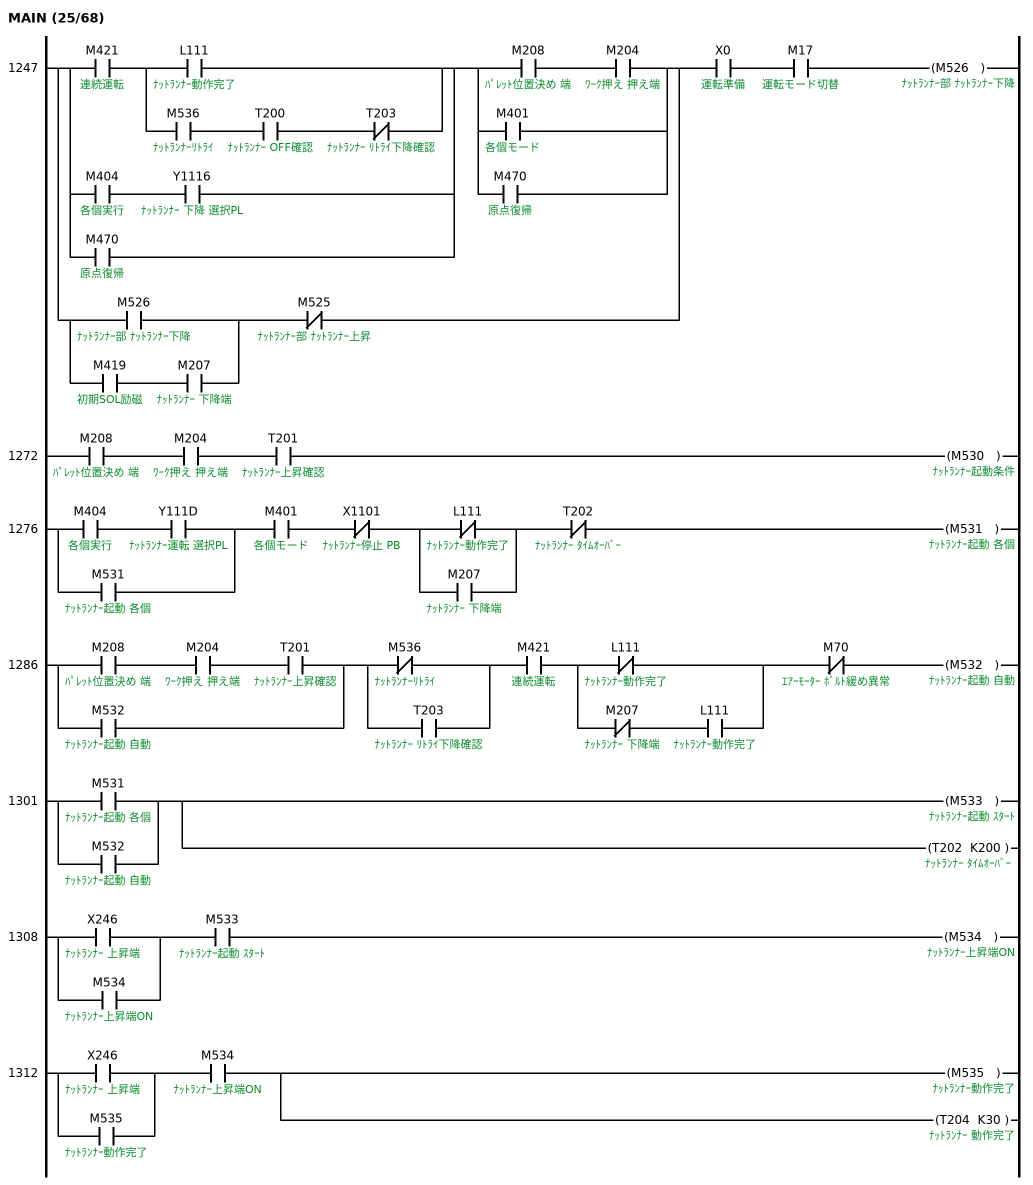
[picture p24: ladder of MAIN, rungs at steps 1247 to 1312]
1247  LD      M421  ; 連続運転
      LD      L111  ; ﾅｯﾄﾗﾝﾅｰ動作完了
      LD      M536  ; ﾅｯﾄﾗﾝﾅｰﾘﾄﾗｲ
      AND     T200  ; ﾅｯﾄﾗﾝﾅｰ OFF確認
      ANI     T203  ; ﾅｯﾄﾗﾝﾅｰ ﾘﾄﾗｲ下降確認
      ORB
      ANB
      LD      M404  ; 各個実行
      AND     Y1116  ; ﾅｯﾄﾗﾝﾅｰ 下降 選択PL
      ORB
      OR      M470  ; 原点復帰
      LD      M208  ; ﾊﾟﾚｯﾄ位置決め 端
      AND     M204  ; ﾜｰｸ押え 押え端
      OR      M401  ; 各個モード
      OR      M470  ; 原点復帰
      ANB
      LD      M526  ; ﾅｯﾄﾗﾝﾅｰ部 ﾅｯﾄﾗﾝﾅｰ下降
      LD      M419  ; 初期SOL励磁
      AND     M207  ; ﾅｯﾄﾗﾝﾅｰ 下降端
      ORB
      ANI     M525  ; ﾅｯﾄﾗﾝﾅｰ部 ﾅｯﾄﾗﾝﾅｰ上昇
      ORB
      AND     X0  ; 運転準備
      AND     M17  ; 運転モード切替
      OUT     M526  ; ﾅｯﾄﾗﾝﾅｰ部 ﾅｯﾄﾗﾝﾅｰ下降
1272  LD      M208  ; ﾊﾟﾚｯﾄ位置決め 端
      AND     M204  ; ﾜｰｸ押え 押え端
      AND     T201  ; ﾅｯﾄﾗﾝﾅｰ上昇確認
      OUT     M530  ; ﾅｯﾄﾗﾝﾅｰ起動条件
1276  LD      M404  ; 各個実行
      AND     Y111D  ; ﾅｯﾄﾗﾝﾅｰ運転 選択PL
      OR      M531  ; ﾅｯﾄﾗﾝﾅｰ起動 各個
      AND     M401  ; 各個モード
      ANI     X1101  ; ﾅｯﾄﾗﾝﾅｰ停止 PB
      LDI     L111  ; ﾅｯﾄﾗﾝﾅｰ動作完了
      OR      M207  ; ﾅｯﾄﾗﾝﾅｰ 下降端
      ANB
      ANI     T202  ; ﾅｯﾄﾗﾝﾅｰ ﾀｲﾑｵｰﾊﾞｰ
      OUT     M531  ; ﾅｯﾄﾗﾝﾅｰ起動 各個
1286  LD      M208  ; ﾊﾟﾚｯﾄ位置決め 端
      AND     M204  ; ﾜｰｸ押え 押え端
      AND     T201  ; ﾅｯﾄﾗﾝﾅｰ上昇確認
      OR      M532  ; ﾅｯﾄﾗﾝﾅｰ起動 自動
      LDI     M536  ; ﾅｯﾄﾗﾝﾅｰﾘﾄﾗｲ
      OR      T203  ; ﾅｯﾄﾗﾝﾅｰ ﾘﾄﾗｲ下降確認
      ANB
      AND     M421  ; 連続運転
      LDI     L111  ; ﾅｯﾄﾗﾝﾅｰ動作完了
      LDI     M207  ; ﾅｯﾄﾗﾝﾅｰ 下降端
      AND     L111  ; ﾅｯﾄﾗﾝﾅｰ動作完了
      ORB
      ANB
      ANI     M70  ; ｴｱｰﾓｰﾀｰ ﾎﾞﾙﾄ緩め異常
      OUT     M532  ; ﾅｯﾄﾗﾝﾅｰ起動 自動
1301  LD      M531  ; ﾅｯﾄﾗﾝﾅｰ起動 各個
      OR      M532  ; ﾅｯﾄﾗﾝﾅｰ起動 自動
      OUT     M533  ; ﾅｯﾄﾗﾝﾅｰ起動 ｽﾀｰﾄ
      OUT     T202 K200  ; ﾅｯﾄﾗﾝﾅｰ ﾀｲﾑｵｰﾊﾞｰ
1308  LD      X246  ; ﾅｯﾄﾗﾝﾅｰ 上昇端
      OR      M534  ; ﾅｯﾄﾗﾝﾅｰ上昇端ON
      AND     M533  ; ﾅｯﾄﾗﾝﾅｰ起動 ｽﾀｰﾄ
      OUT     M534  ; ﾅｯﾄﾗﾝﾅｰ上昇端ON
1312  LD      X246  ; ﾅｯﾄﾗﾝﾅｰ 上昇端
      OR      M535  ; ﾅｯﾄﾗﾝﾅｰ動作完了
      AND     M534  ; ﾅｯﾄﾗﾝﾅｰ上昇端ON
      OUT     M535  ; ﾅｯﾄﾗﾝﾅｰ動作完了
      OUT     T204 K30  ; ﾅｯﾄﾗﾝﾅｰ 動作完了
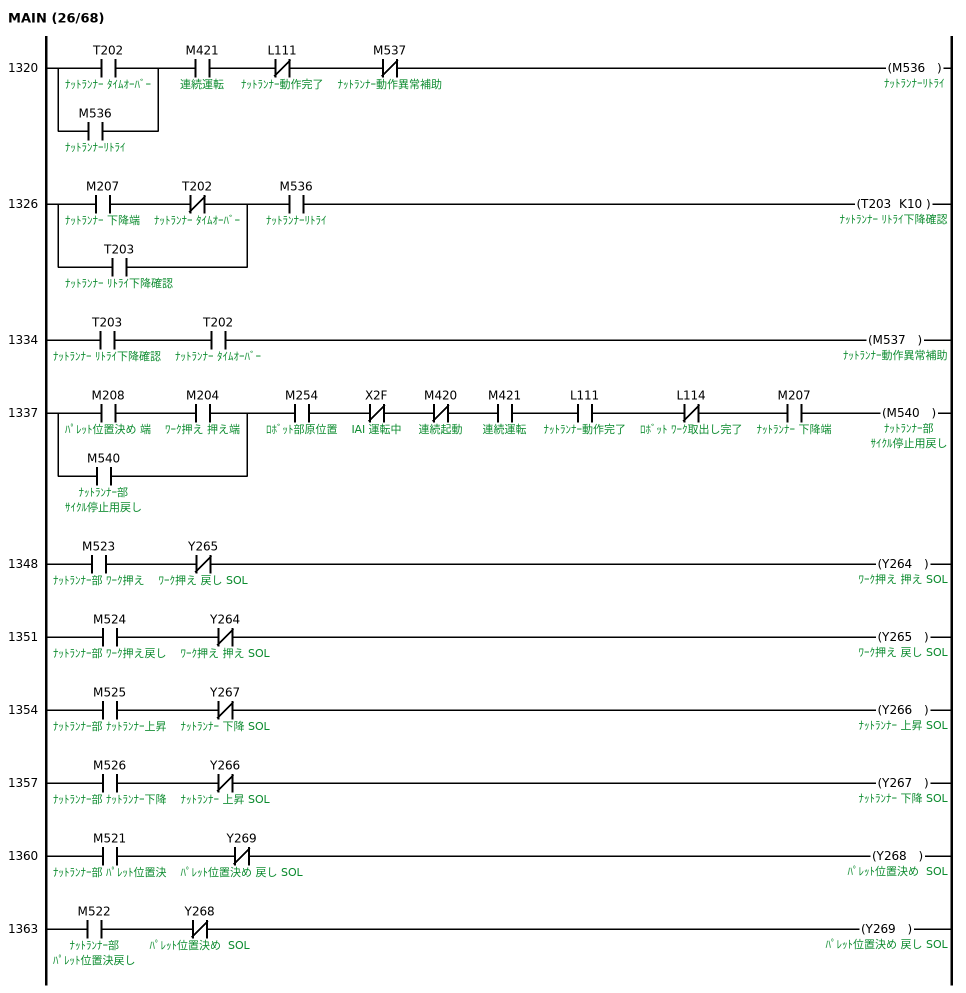
1320  LD      T202  ; ﾅｯﾄﾗﾝﾅｰ ﾀｲﾑｵｰﾊﾞｰ
      OR      M536  ; ﾅｯﾄﾗﾝﾅｰﾘﾄﾗｲ
      AND     M421  ; 連続運転
      ANI     L111  ; ﾅｯﾄﾗﾝﾅｰ動作完了
      ANI     M537  ; ﾅｯﾄﾗﾝﾅｰ動作異常補助
      OUT     M536  ; ﾅｯﾄﾗﾝﾅｰﾘﾄﾗｲ
1326  LD      M207  ; ﾅｯﾄﾗﾝﾅｰ 下降端
      ANI     T202  ; ﾅｯﾄﾗﾝﾅｰ ﾀｲﾑｵｰﾊﾞｰ
      OR      T203  ; ﾅｯﾄﾗﾝﾅｰ ﾘﾄﾗｲ下降確認
      AND     M536  ; ﾅｯﾄﾗﾝﾅｰﾘﾄﾗｲ
      OUT     T203 K10  ; ﾅｯﾄﾗﾝﾅｰ ﾘﾄﾗｲ下降確認
1334  LD      T203  ; ﾅｯﾄﾗﾝﾅｰ ﾘﾄﾗｲ下降確認
      AND     T202  ; ﾅｯﾄﾗﾝﾅｰ ﾀｲﾑｵｰﾊﾞｰ
      OUT     M537  ; ﾅｯﾄﾗﾝﾅｰ動作異常補助
1337  LD      M208  ; ﾊﾟﾚｯﾄ位置決め 端
      AND     M204  ; ﾜｰｸ押え 押え端
      OR      M540  ; ﾅｯﾄﾗﾝﾅｰ部 ｻｲｸﾙ停止用戻し
      AND     M254  ; ﾛﾎﾞｯﾄ部原位置
      ANI     X2F  ; IAI 運転中
      ANI     M420  ; 連続起動
      AND     M421  ; 連続運転
      AND     L111  ; ﾅｯﾄﾗﾝﾅｰ動作完了
      ANI     L114  ; ﾛﾎﾞｯﾄ ﾜｰｸ取出し完了
      AND     M207  ; ﾅｯﾄﾗﾝﾅｰ 下降端
      OUT     M540  ; ﾅｯﾄﾗﾝﾅｰ部 ｻｲｸﾙ停止用戻し
1348  LD      M523  ; ﾅｯﾄﾗﾝﾅｰ部 ﾜｰｸ押え
      ANI     Y265  ; ﾜｰｸ押え 戻し SOL
      OUT     Y264  ; ﾜｰｸ押え 押え SOL
1351  LD      M524  ; ﾅｯﾄﾗﾝﾅｰ部 ﾜｰｸ押え戻し
      ANI     Y264  ; ﾜｰｸ押え 押え SOL
      OUT     Y265  ; ﾜｰｸ押え 戻し SOL
1354  LD      M525  ; ﾅｯﾄﾗﾝﾅｰ部 ﾅｯﾄﾗﾝﾅｰ上昇
      ANI     Y267  ; ﾅｯﾄﾗﾝﾅｰ 下降 SOL
      OUT     Y266  ; ﾅｯﾄﾗﾝﾅｰ 上昇 SOL
1357  LD      M526  ; ﾅｯﾄﾗﾝﾅｰ部 ﾅｯﾄﾗﾝﾅｰ下降
      ANI     Y266  ; ﾅｯﾄﾗﾝﾅｰ 上昇 SOL
      OUT     Y267  ; ﾅｯﾄﾗﾝﾅｰ 下降 SOL
1360  LD      M521  ; ﾅｯﾄﾗﾝﾅｰ部 ﾊﾟﾚｯﾄ位置決
      ANI     Y269  ; ﾊﾟﾚｯﾄ位置決め 戻し SOL
      OUT     Y268  ; ﾊﾟﾚｯﾄ位置決め  SOL
1363  LD      M522  ; ﾅｯﾄﾗﾝﾅｰ部 ﾊﾟﾚｯﾄ位置決戻し
      ANI     Y268  ; ﾊﾟﾚｯﾄ位置決め  SOL
      OUT     Y269  ; ﾊﾟﾚｯﾄ位置決め 戻し SOL
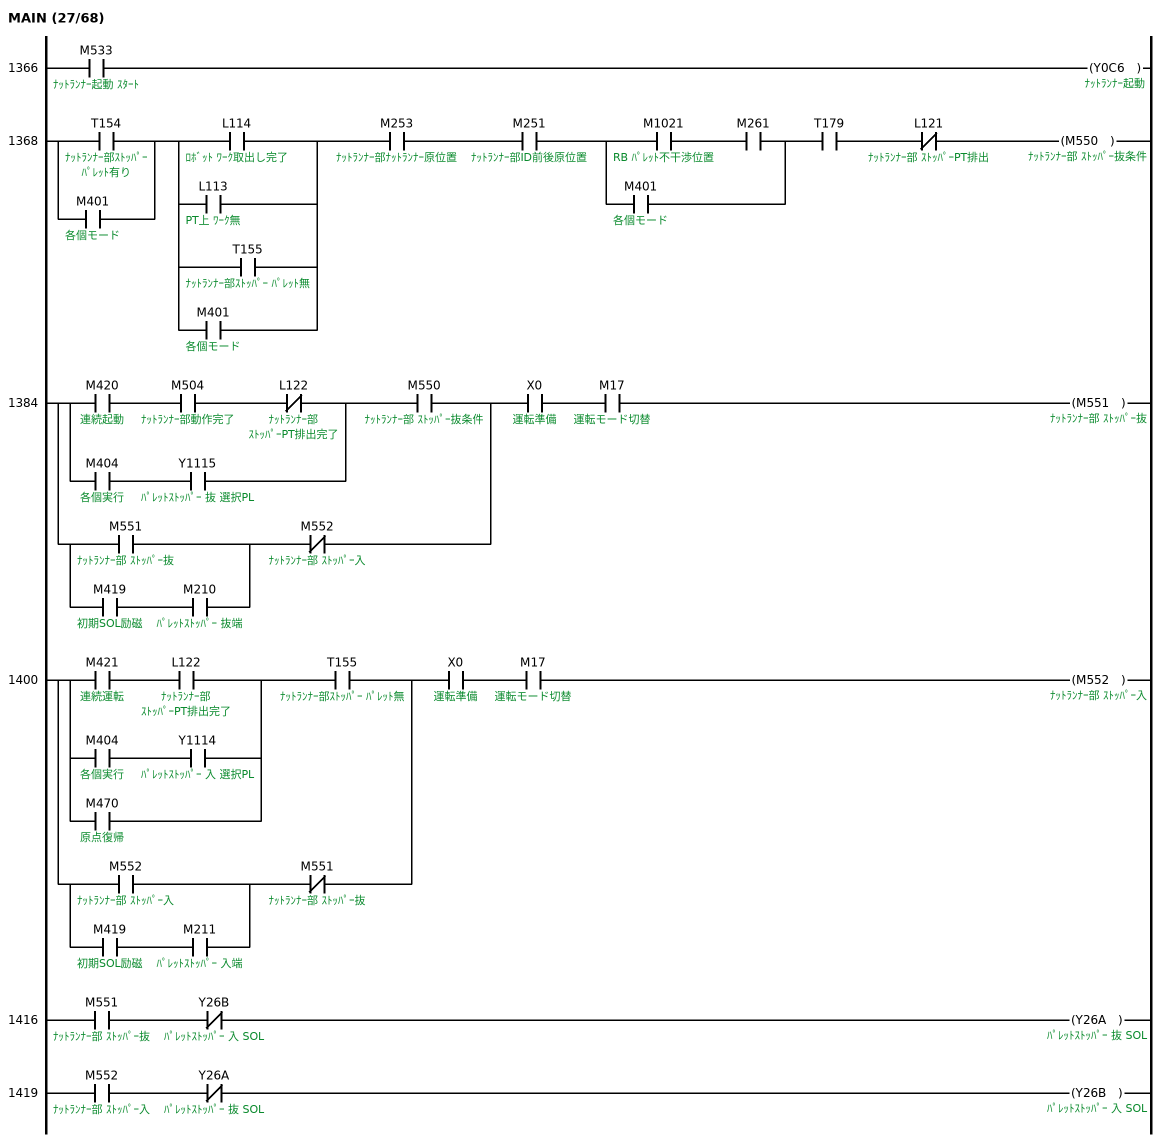
1366  LD      M533  ; ﾅｯﾄﾗﾝﾅｰ起動 ｽﾀｰﾄ
      OUT     Y0C6  ; ﾅｯﾄﾗﾝﾅｰ起動
1368  LD      T154  ; ﾅｯﾄﾗﾝﾅｰ部ｽﾄｯﾊﾟｰ ﾊﾟﾚｯﾄ有り
      OR      M401  ; 各個モード
      LD      L114  ; ﾛﾎﾞｯﾄ ﾜｰｸ取出し完了
      OR      L113  ; PT上 ﾜｰｸ無
      OR      T155  ; ﾅｯﾄﾗﾝﾅｰ部ｽﾄｯﾊﾟｰ ﾊﾟﾚｯﾄ無
      OR      M401  ; 各個モード
      ANB
      AND     M253  ; ﾅｯﾄﾗﾝﾅｰ部ﾅｯﾄﾗﾝﾅｰ原位置
      AND     M251  ; ﾅｯﾄﾗﾝﾅｰ部ID前後原位置
      LD      M1021  ; RB ﾊﾟﾚｯﾄ不干渉位置
      AND     M261
      OR      M401  ; 各個モード
      ANB
      AND     T179
      ANI     L121  ; ﾅｯﾄﾗﾝﾅｰ部 ｽﾄｯﾊﾟｰPT排出
      OUT     M550  ; ﾅｯﾄﾗﾝﾅｰ部 ｽﾄｯﾊﾟｰ抜条件
1384  LD      M420  ; 連続起動
      AND     M504  ; ﾅｯﾄﾗﾝﾅｰ部動作完了
      ANI     L122  ; ﾅｯﾄﾗﾝﾅｰ部 ｽﾄｯﾊﾟｰPT排出完了
      LD      M404  ; 各個実行
      AND     Y1115  ; ﾊﾟﾚｯﾄｽﾄｯﾊﾟｰ 抜 選択PL
      ORB
      AND     M550  ; ﾅｯﾄﾗﾝﾅｰ部 ｽﾄｯﾊﾟｰ抜条件
      LD      M551  ; ﾅｯﾄﾗﾝﾅｰ部 ｽﾄｯﾊﾟｰ抜
      LD      M419  ; 初期SOL励磁
      AND     M210  ; ﾊﾟﾚｯﾄｽﾄｯﾊﾟｰ 抜端
      ORB
      ANI     M552  ; ﾅｯﾄﾗﾝﾅｰ部 ｽﾄｯﾊﾟｰ入
      ORB
      AND     X0  ; 運転準備
      AND     M17  ; 運転モード切替
      OUT     M551  ; ﾅｯﾄﾗﾝﾅｰ部 ｽﾄｯﾊﾟｰ抜
1400  LD      M421  ; 連続運転
      AND     L122  ; ﾅｯﾄﾗﾝﾅｰ部 ｽﾄｯﾊﾟｰPT排出完了
      LD      M404  ; 各個実行
      AND     Y1114  ; ﾊﾟﾚｯﾄｽﾄｯﾊﾟｰ 入 選択PL
      ORB
      OR      M470  ; 原点復帰
      AND     T155  ; ﾅｯﾄﾗﾝﾅｰ部ｽﾄｯﾊﾟｰ ﾊﾟﾚｯﾄ無
      LD      M552  ; ﾅｯﾄﾗﾝﾅｰ部 ｽﾄｯﾊﾟｰ入
      LD      M419  ; 初期SOL励磁
      AND     M211  ; ﾊﾟﾚｯﾄｽﾄｯﾊﾟｰ 入端
      ORB
      ANI     M551  ; ﾅｯﾄﾗﾝﾅｰ部 ｽﾄｯﾊﾟｰ抜
      ORB
      AND     X0  ; 運転準備
      AND     M17  ; 運転モード切替
      OUT     M552  ; ﾅｯﾄﾗﾝﾅｰ部 ｽﾄｯﾊﾟｰ入
1416  LD      M551  ; ﾅｯﾄﾗﾝﾅｰ部 ｽﾄｯﾊﾟｰ抜
      ANI     Y26B  ; ﾊﾟﾚｯﾄｽﾄｯﾊﾟｰ 入 SOL
      OUT     Y26A  ; ﾊﾟﾚｯﾄｽﾄｯﾊﾟｰ 抜 SOL
1419  LD      M552  ; ﾅｯﾄﾗﾝﾅｰ部 ｽﾄｯﾊﾟｰ入
      ANI     Y26A  ; ﾊﾟﾚｯﾄｽﾄｯﾊﾟｰ 抜 SOL
      OUT     Y26B  ; ﾊﾟﾚｯﾄｽﾄｯﾊﾟｰ 入 SOL
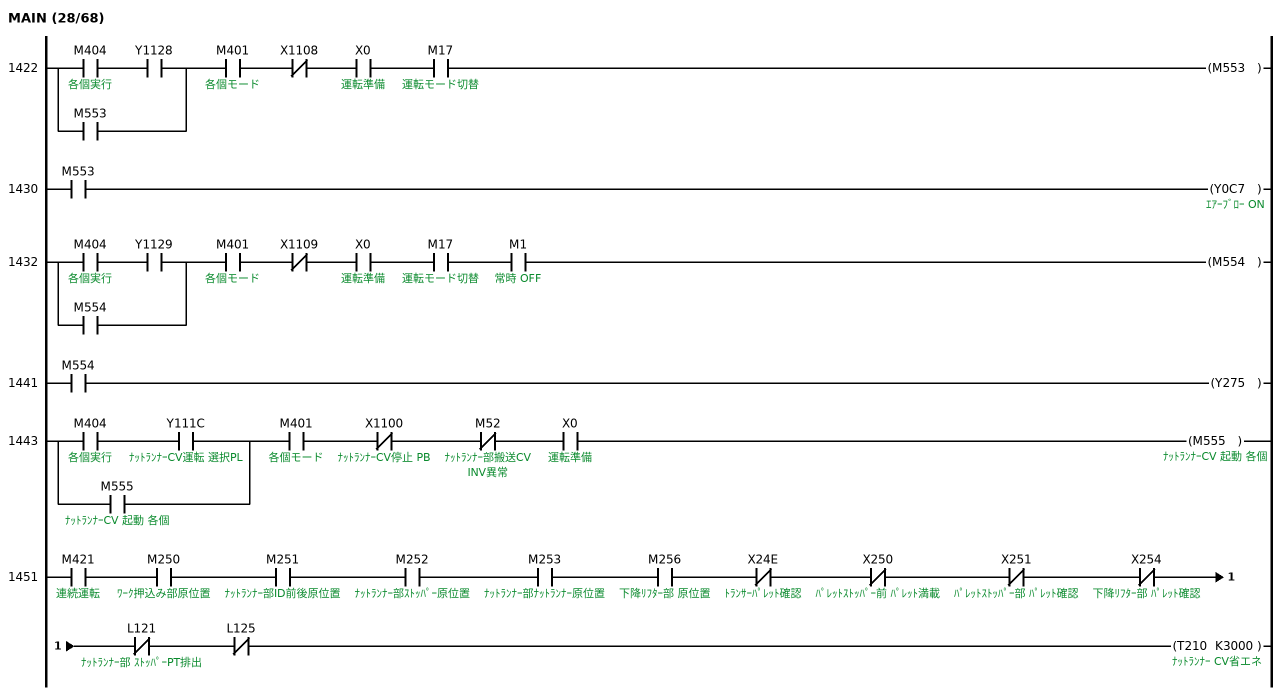
1422  LD      M404  ; 各個実行
      AND     Y1128
      OR      M553
      AND     M401  ; 各個モード
      ANI     X1108
      AND     X0  ; 運転準備
      AND     M17  ; 運転モード切替
      OUT     M553
1430  LD      M553
      OUT     Y0C7  ; ｴｱｰﾌﾞﾛｰ ON
1432  LD      M404  ; 各個実行
      AND     Y1129
      OR      M554
      AND     M401  ; 各個モード
      ANI     X1109
      AND     X0  ; 運転準備
      AND     M17  ; 運転モード切替
      AND     M1  ; 常時 OFF
      OUT     M554
1441  LD      M554
      OUT     Y275
1443  LD      M404  ; 各個実行
      AND     Y111C  ; ﾅｯﾄﾗﾝﾅｰCV運転 選択PL
      OR      M555  ; ﾅｯﾄﾗﾝﾅｰCV 起動 各個
      AND     M401  ; 各個モード
      ANI     X1100  ; ﾅｯﾄﾗﾝﾅｰCV停止 PB
      ANI     M52  ; ﾅｯﾄﾗﾝﾅｰ部搬送CV INV異常
      AND     X0  ; 運転準備
      OUT     M555  ; ﾅｯﾄﾗﾝﾅｰCV 起動 各個
1451  LD      M421  ; 連続運転
      AND     M250  ; ﾜｰｸ押込み部原位置
      AND     M251  ; ﾅｯﾄﾗﾝﾅｰ部ID前後原位置
      AND     M252  ; ﾅｯﾄﾗﾝﾅｰ部ｽﾄｯﾊﾟｰ原位置
      AND     M253  ; ﾅｯﾄﾗﾝﾅｰ部ﾅｯﾄﾗﾝﾅｰ原位置
      AND     M256  ; 下降ﾘﾌﾀｰ部 原位置
      ANI     X24E  ; ﾄﾗﾝｻｰﾊﾟﾚｯﾄ確認
      ANI     X250  ; ﾊﾟﾚｯﾄｽﾄｯﾊﾟｰ前 ﾊﾟﾚｯﾄ満載
      ANI     X251  ; ﾊﾟﾚｯﾄｽﾄｯﾊﾟｰ部 ﾊﾟﾚｯﾄ確認
      ANI     X254  ; 下降ﾘﾌﾀｰ部 ﾊﾟﾚｯﾄ確認
      ANI     L121  ; ﾅｯﾄﾗﾝﾅｰ部 ｽﾄｯﾊﾟｰPT排出
      ANI     L125
      OUT     T210 K3000  ; ﾅｯﾄﾗﾝﾅｰ CV省エネ
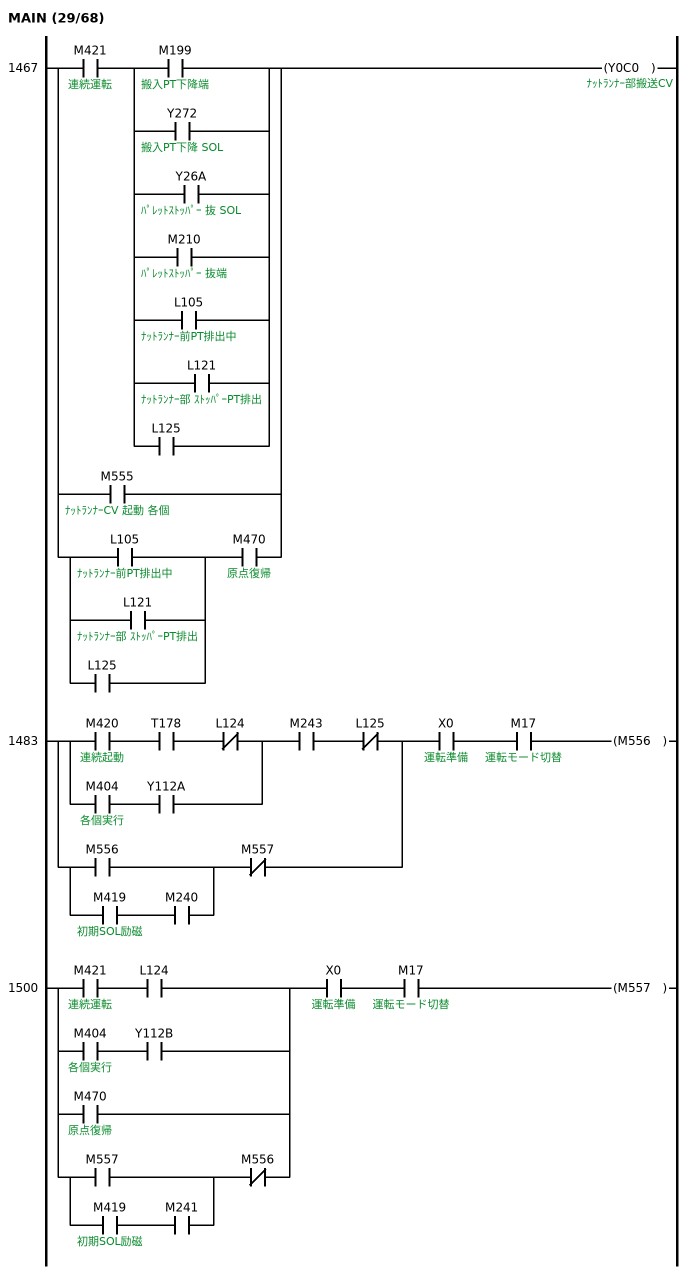
1467  LD      M421  ; 連続運転
      LD      M199  ; 搬入PT下降端
      OR      Y272  ; 搬入PT下降 SOL
      OR      Y26A  ; ﾊﾟﾚｯﾄｽﾄｯﾊﾟｰ 抜 SOL
      OR      M210  ; ﾊﾟﾚｯﾄｽﾄｯﾊﾟｰ 抜端
      OR      L105  ; ﾅｯﾄﾗﾝﾅｰ前PT排出中
      OR      L121  ; ﾅｯﾄﾗﾝﾅｰ部 ｽﾄｯﾊﾟｰPT排出
      OR      L125
      ANB
      OR      M555  ; ﾅｯﾄﾗﾝﾅｰCV 起動 各個
      LD      L105  ; ﾅｯﾄﾗﾝﾅｰ前PT排出中
      OR      L121  ; ﾅｯﾄﾗﾝﾅｰ部 ｽﾄｯﾊﾟｰPT排出
      OR      L125
      AND     M470  ; 原点復帰
      ORB
      OUT     Y0C0  ; ﾅｯﾄﾗﾝﾅｰ部搬送CV
1483  LD      M420  ; 連続起動
      AND     T178
      ANI     L124
      LD      M404  ; 各個実行
      AND     Y112A
      ORB
      AND     M243
      ANI     L125
      LD      M556
      LD      M419  ; 初期SOL励磁
      AND     M240
      ORB
      ANI     M557
      ORB
      AND     X0  ; 運転準備
      AND     M17  ; 運転モード切替
      OUT     M556
1500  LD      M421  ; 連続運転
      AND     L124
      LD      M404  ; 各個実行
      AND     Y112B
      ORB
      OR      M470  ; 原点復帰
      LD      M557
      LD      M419  ; 初期SOL励磁
      AND     M241
      ORB
      ANI     M556
      ORB
      AND     X0  ; 運転準備
      AND     M17  ; 運転モード切替
      OUT     M557
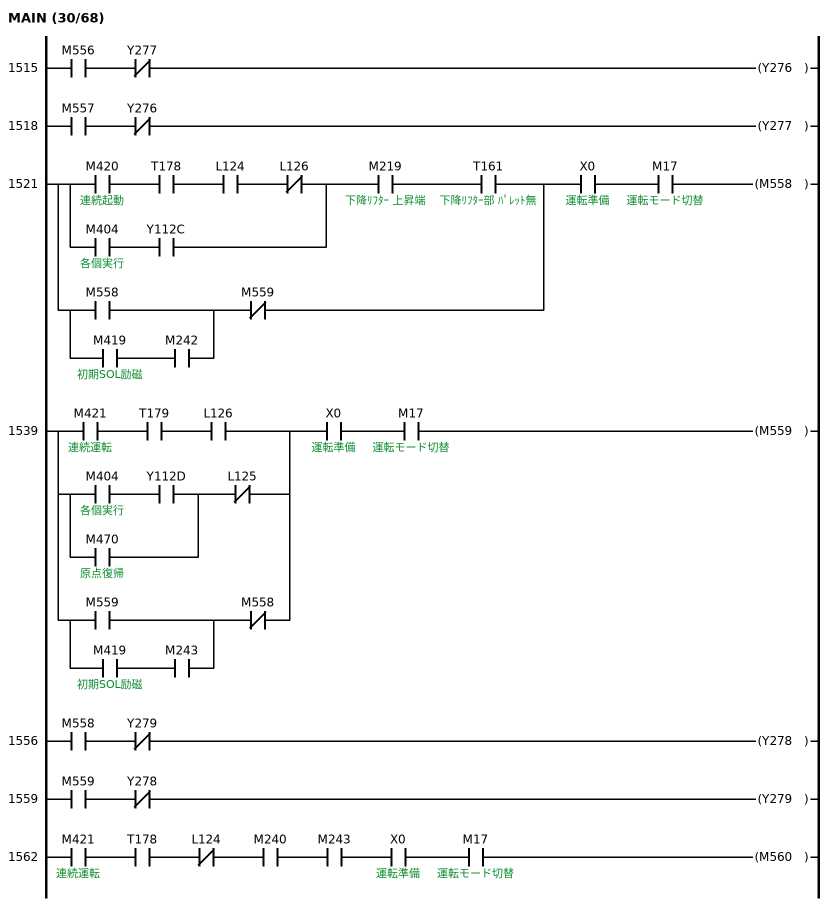
1515  LD      M556
      ANI     Y277
      OUT     Y276
1518  LD      M557
      ANI     Y276
      OUT     Y277
1521  LD      M420  ; 連続起動
      AND     T178
      AND     L124
      ANI     L126
      LD      M404  ; 各個実行
      AND     Y112C
      ORB
      AND     M219  ; 下降ﾘﾌﾀｰ 上昇端
      AND     T161  ; 下降ﾘﾌﾀｰ部 ﾊﾟﾚｯﾄ無
      LD      M558
      LD      M419  ; 初期SOL励磁
      AND     M242
      ORB
      ANI     M559
      ORB
      AND     X0  ; 運転準備
      AND     M17  ; 運転モード切替
      OUT     M558
1539  LD      M421  ; 連続運転
      AND     T179
      AND     L126
      LD      M404  ; 各個実行
      AND     Y112D
      OR      M470  ; 原点復帰
      ANI     L125
      ORB
      LD      M559
      LD      M419  ; 初期SOL励磁
      AND     M243
      ORB
      ANI     M558
      ORB
      AND     X0  ; 運転準備
      AND     M17  ; 運転モード切替
      OUT     M559
1556  LD      M558
      ANI     Y279
      OUT     Y278
1559  LD      M559
      ANI     Y278
      OUT     Y279
1562  LD      M421  ; 連続運転
      AND     T178
      ANI     L124
      AND     M240
      AND     M243
      AND     X0  ; 運転準備
      AND     M17  ; 運転モード切替
      OUT     M560
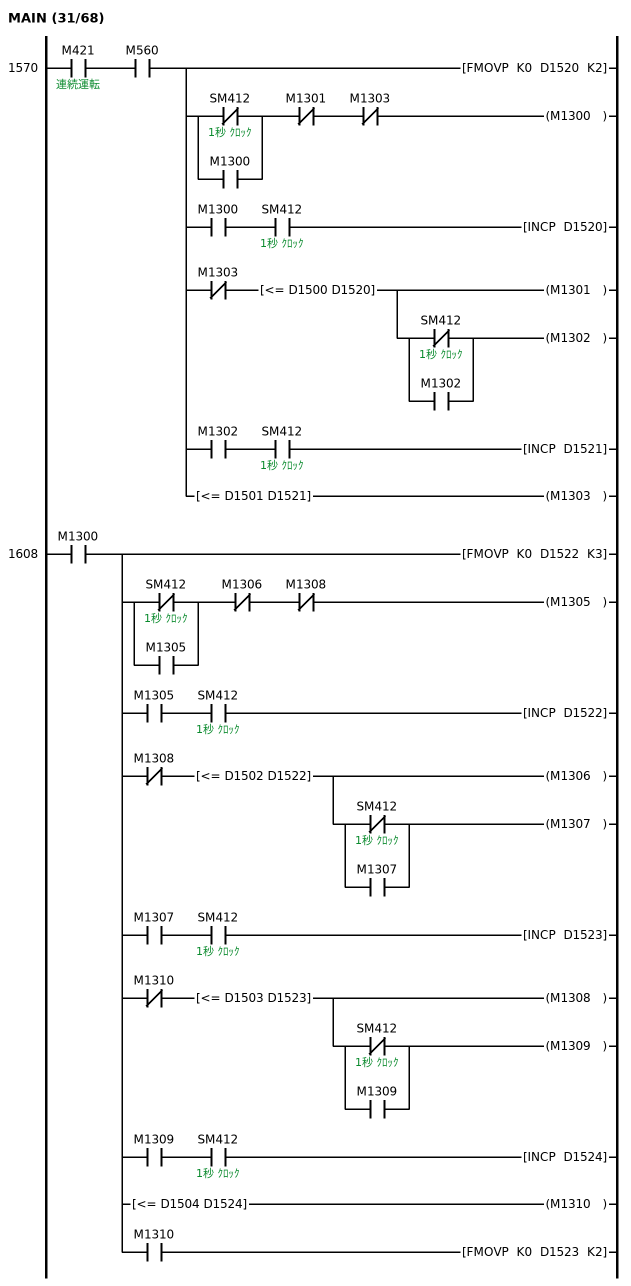
1570  LD      M421  ; 連続運転
      AND     M560
      FMOVP   K0 D1520 K2
      MPS
      LDI     SM412  ; 1秒 ｸﾛｯｸ
      OR      M1300
      ANB
      ANI     M1301
      ANI     M1303
      OUT     M1300
      MRD
      AND     M1300
      AND     SM412  ; 1秒 ｸﾛｯｸ
      INCP    D1520
      MRD
      ANI     M1303
      AND<=   D1500 D1520
      OUT     M1301
      LDI     SM412  ; 1秒 ｸﾛｯｸ
      OR      M1302
      ANB
      OUT     M1302
      MRD
      AND     M1302
      AND     SM412  ; 1秒 ｸﾛｯｸ
      INCP    D1521
      MPP
      AND<=   D1501 D1521
      OUT     M1303
1608  LD      M1300
      FMOVP   K0 D1522 K3
      MPS
      LDI     SM412  ; 1秒 ｸﾛｯｸ
      OR      M1305
      ANB
      ANI     M1306
      ANI     M1308
      OUT     M1305
      MRD
      AND     M1305
      AND     SM412  ; 1秒 ｸﾛｯｸ
      INCP    D1522
      MRD
      ANI     M1308
      AND<=   D1502 D1522
      OUT     M1306
      LDI     SM412  ; 1秒 ｸﾛｯｸ
      OR      M1307
      ANB
      OUT     M1307
      MRD
      AND     M1307
      AND     SM412  ; 1秒 ｸﾛｯｸ
      INCP    D1523
      MRD
      ANI     M1310
      AND<=   D1503 D1523
      OUT     M1308
      LDI     SM412  ; 1秒 ｸﾛｯｸ
      OR      M1309
      ANB
      OUT     M1309
      MRD
      AND     M1309
      AND     SM412  ; 1秒 ｸﾛｯｸ
      INCP    D1524
      MRD
      AND<=   D1504 D1524
      OUT     M1310
      MPP
      AND     M1310
      FMOVP   K0 D1523 K2
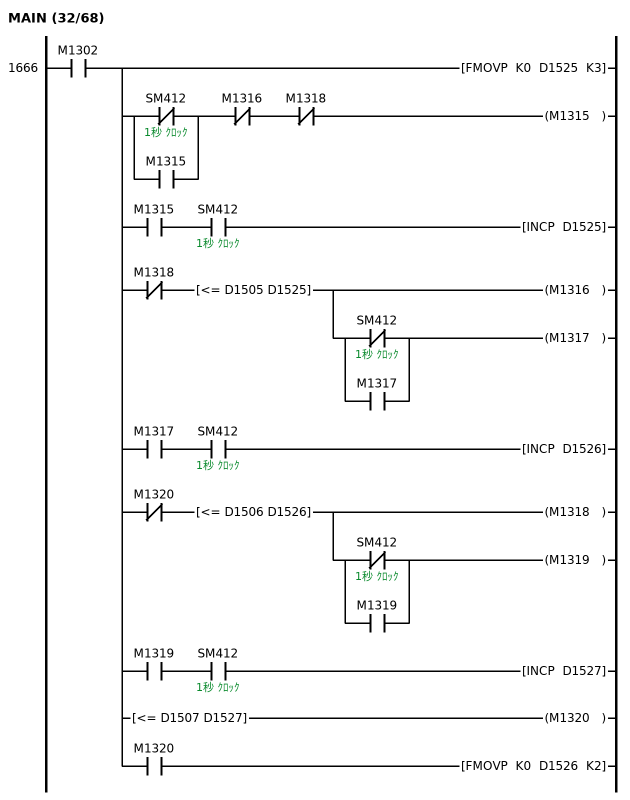
1666  LD      M1302
      FMOVP   K0 D1525 K3
      MPS
      LDI     SM412  ; 1秒 ｸﾛｯｸ
      OR      M1315
      ANB
      ANI     M1316
      ANI     M1318
      OUT     M1315
      MRD
      AND     M1315
      AND     SM412  ; 1秒 ｸﾛｯｸ
      INCP    D1525
      MRD
      ANI     M1318
      AND<=   D1505 D1525
      OUT     M1316
      LDI     SM412  ; 1秒 ｸﾛｯｸ
      OR      M1317
      ANB
      OUT     M1317
      MRD
      AND     M1317
      AND     SM412  ; 1秒 ｸﾛｯｸ
      INCP    D1526
      MRD
      ANI     M1320
      AND<=   D1506 D1526
      OUT     M1318
      LDI     SM412  ; 1秒 ｸﾛｯｸ
      OR      M1319
      ANB
      OUT     M1319
      MRD
      AND     M1319
      AND     SM412  ; 1秒 ｸﾛｯｸ
      INCP    D1527
      MRD
      AND<=   D1507 D1527
      OUT     M1320
      MPP
      AND     M1320
      FMOVP   K0 D1526 K2
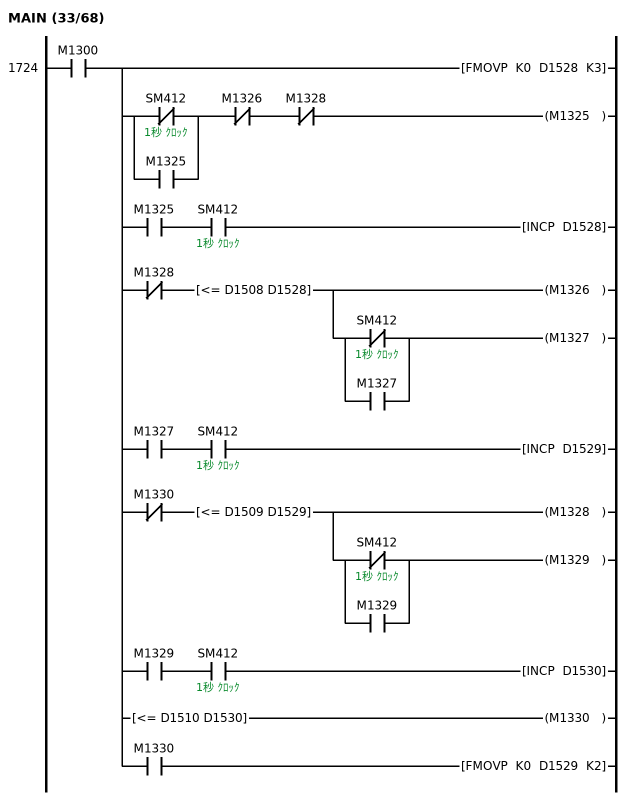
1724  LD      M1300
      FMOVP   K0 D1528 K3
      MPS
      LDI     SM412  ; 1秒 ｸﾛｯｸ
      OR      M1325
      ANB
      ANI     M1326
      ANI     M1328
      OUT     M1325
      MRD
      AND     M1325
      AND     SM412  ; 1秒 ｸﾛｯｸ
      INCP    D1528
      MRD
      ANI     M1328
      AND<=   D1508 D1528
      OUT     M1326
      LDI     SM412  ; 1秒 ｸﾛｯｸ
      OR      M1327
      ANB
      OUT     M1327
      MRD
      AND     M1327
      AND     SM412  ; 1秒 ｸﾛｯｸ
      INCP    D1529
      MRD
      ANI     M1330
      AND<=   D1509 D1529
      OUT     M1328
      LDI     SM412  ; 1秒 ｸﾛｯｸ
      OR      M1329
      ANB
      OUT     M1329
      MRD
      AND     M1329
      AND     SM412  ; 1秒 ｸﾛｯｸ
      INCP    D1530
      MRD
      AND<=   D1510 D1530
      OUT     M1330
      MPP
      AND     M1330
      FMOVP   K0 D1529 K2
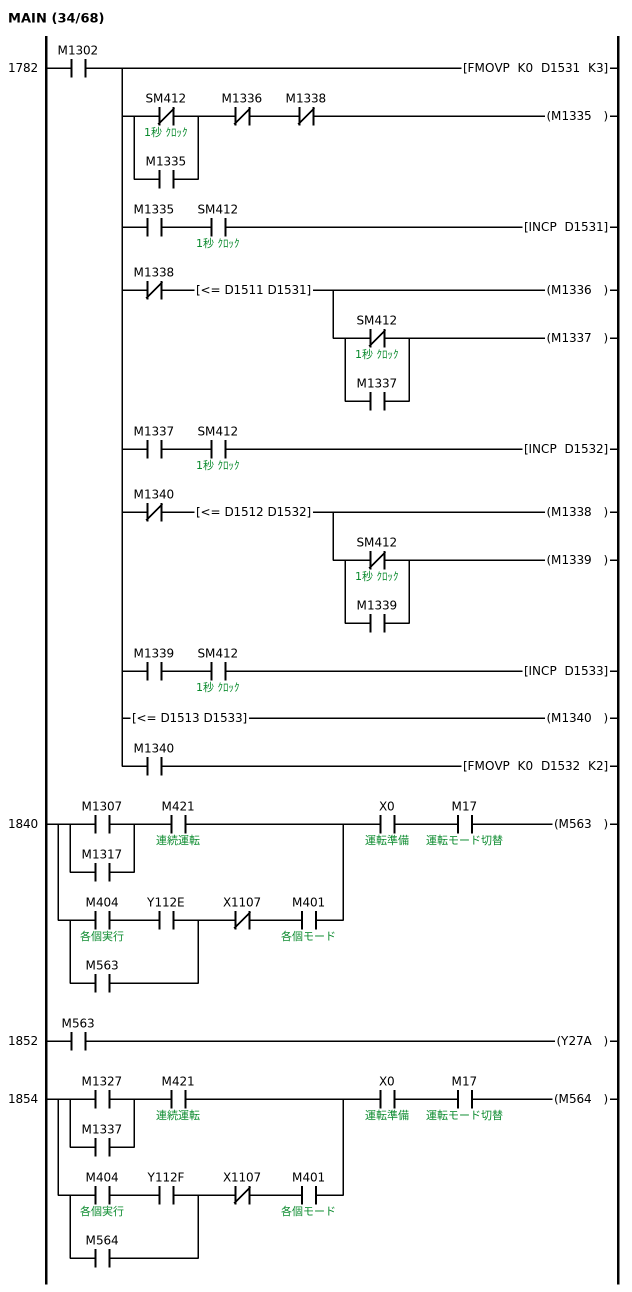
1782  LD      M1302
      FMOVP   K0 D1531 K3
      MPS
      LDI     SM412  ; 1秒 ｸﾛｯｸ
      OR      M1335
      ANB
      ANI     M1336
      ANI     M1338
      OUT     M1335
      MRD
      AND     M1335
      AND     SM412  ; 1秒 ｸﾛｯｸ
      INCP    D1531
      MRD
      ANI     M1338
      AND<=   D1511 D1531
      OUT     M1336
      LDI     SM412  ; 1秒 ｸﾛｯｸ
      OR      M1337
      ANB
      OUT     M1337
      MRD
      AND     M1337
      AND     SM412  ; 1秒 ｸﾛｯｸ
      INCP    D1532
      MRD
      ANI     M1340
      AND<=   D1512 D1532
      OUT     M1338
      LDI     SM412  ; 1秒 ｸﾛｯｸ
      OR      M1339
      ANB
      OUT     M1339
      MRD
      AND     M1339
      AND     SM412  ; 1秒 ｸﾛｯｸ
      INCP    D1533
      MRD
      AND<=   D1513 D1533
      OUT     M1340
      MPP
      AND     M1340
      FMOVP   K0 D1532 K2
1840  LD      M1307
      OR      M1317
      AND     M421  ; 連続運転
      LD      M404  ; 各個実行
      AND     Y112E
      OR      M563
      ANI     X1107
      AND     M401  ; 各個モード
      ORB
      AND     X0  ; 運転準備
      AND     M17  ; 運転モード切替
      OUT     M563
1852  LD      M563
      OUT     Y27A
1854  LD      M1327
      OR      M1337
      AND     M421  ; 連続運転
      LD      M404  ; 各個実行
      AND     Y112F
      OR      M564
      ANI     X1107
      AND     M401  ; 各個モード
      ORB
      AND     X0  ; 運転準備
      AND     M17  ; 運転モード切替
      OUT     M564
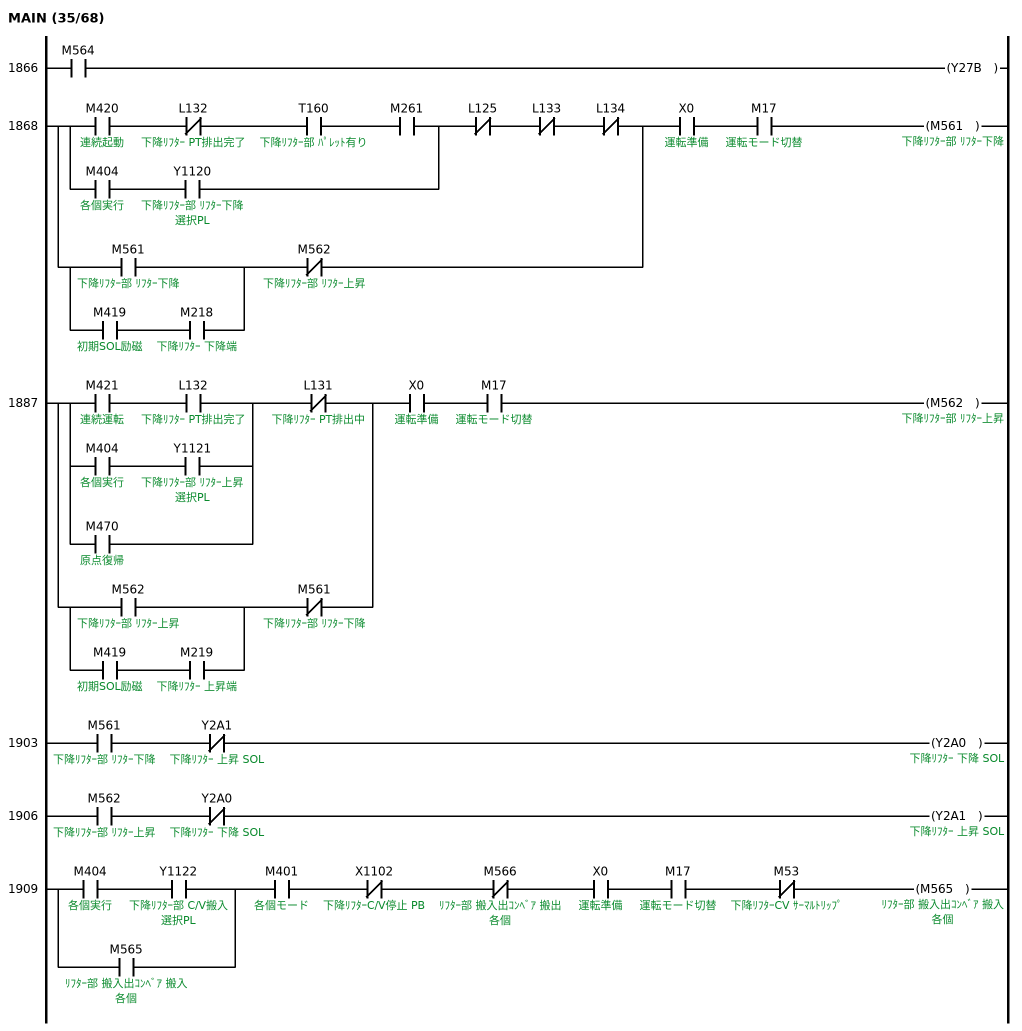
1866  LD      M564
      OUT     Y27B
1868  LD      M420  ; 連続起動
      ANI     L132  ; 下降ﾘﾌﾀｰ PT排出完了
      AND     T160  ; 下降ﾘﾌﾀｰ部 ﾊﾟﾚｯﾄ有り
      AND     M261
      LD      M404  ; 各個実行
      AND     Y1120  ; 下降ﾘﾌﾀｰ部 ﾘﾌﾀｰ下降 選択PL
      ORB
      ANI     L125
      ANI     L133
      ANI     L134
      LD      M561  ; 下降ﾘﾌﾀｰ部 ﾘﾌﾀｰ下降
      LD      M419  ; 初期SOL励磁
      AND     M218  ; 下降ﾘﾌﾀｰ 下降端
      ORB
      ANI     M562  ; 下降ﾘﾌﾀｰ部 ﾘﾌﾀｰ上昇
      ORB
      AND     X0  ; 運転準備
      AND     M17  ; 運転モード切替
      OUT     M561  ; 下降ﾘﾌﾀｰ部 ﾘﾌﾀｰ下降
1887  LD      M421  ; 連続運転
      AND     L132  ; 下降ﾘﾌﾀｰ PT排出完了
      LD      M404  ; 各個実行
      AND     Y1121  ; 下降ﾘﾌﾀｰ部 ﾘﾌﾀｰ上昇 選択PL
      ORB
      OR      M470  ; 原点復帰
      ANI     L131  ; 下降ﾘﾌﾀｰ PT排出中
      LD      M562  ; 下降ﾘﾌﾀｰ部 ﾘﾌﾀｰ上昇
      LD      M419  ; 初期SOL励磁
      AND     M219  ; 下降ﾘﾌﾀｰ 上昇端
      ORB
      ANI     M561  ; 下降ﾘﾌﾀｰ部 ﾘﾌﾀｰ下降
      ORB
      AND     X0  ; 運転準備
      AND     M17  ; 運転モード切替
      OUT     M562  ; 下降ﾘﾌﾀｰ部 ﾘﾌﾀｰ上昇
1903  LD      M561  ; 下降ﾘﾌﾀｰ部 ﾘﾌﾀｰ下降
      ANI     Y2A1  ; 下降ﾘﾌﾀｰ 上昇 SOL
      OUT     Y2A0  ; 下降ﾘﾌﾀｰ 下降 SOL
1906  LD      M562  ; 下降ﾘﾌﾀｰ部 ﾘﾌﾀｰ上昇
      ANI     Y2A0  ; 下降ﾘﾌﾀｰ 下降 SOL
      OUT     Y2A1  ; 下降ﾘﾌﾀｰ 上昇 SOL
1909  LD      M404  ; 各個実行
      AND     Y1122  ; 下降ﾘﾌﾀｰ部 C/V搬入 選択PL
      OR      M565  ; ﾘﾌﾀｰ部 搬入出ｺﾝﾍﾞｱ 搬入 各個
      AND     M401  ; 各個モード
      ANI     X1102  ; 下降ﾘﾌﾀｰC/V停止 PB
      ANI     M566  ; ﾘﾌﾀｰ部 搬入出ｺﾝﾍﾞｱ 搬出 各個
      AND     X0  ; 運転準備
      AND     M17  ; 運転モード切替
      ANI     M53  ; 下降ﾘﾌﾀｰCV ｻｰﾏﾙﾄﾘｯﾌﾟ
      OUT     M565  ; ﾘﾌﾀｰ部 搬入出ｺﾝﾍﾞｱ 搬入 各個
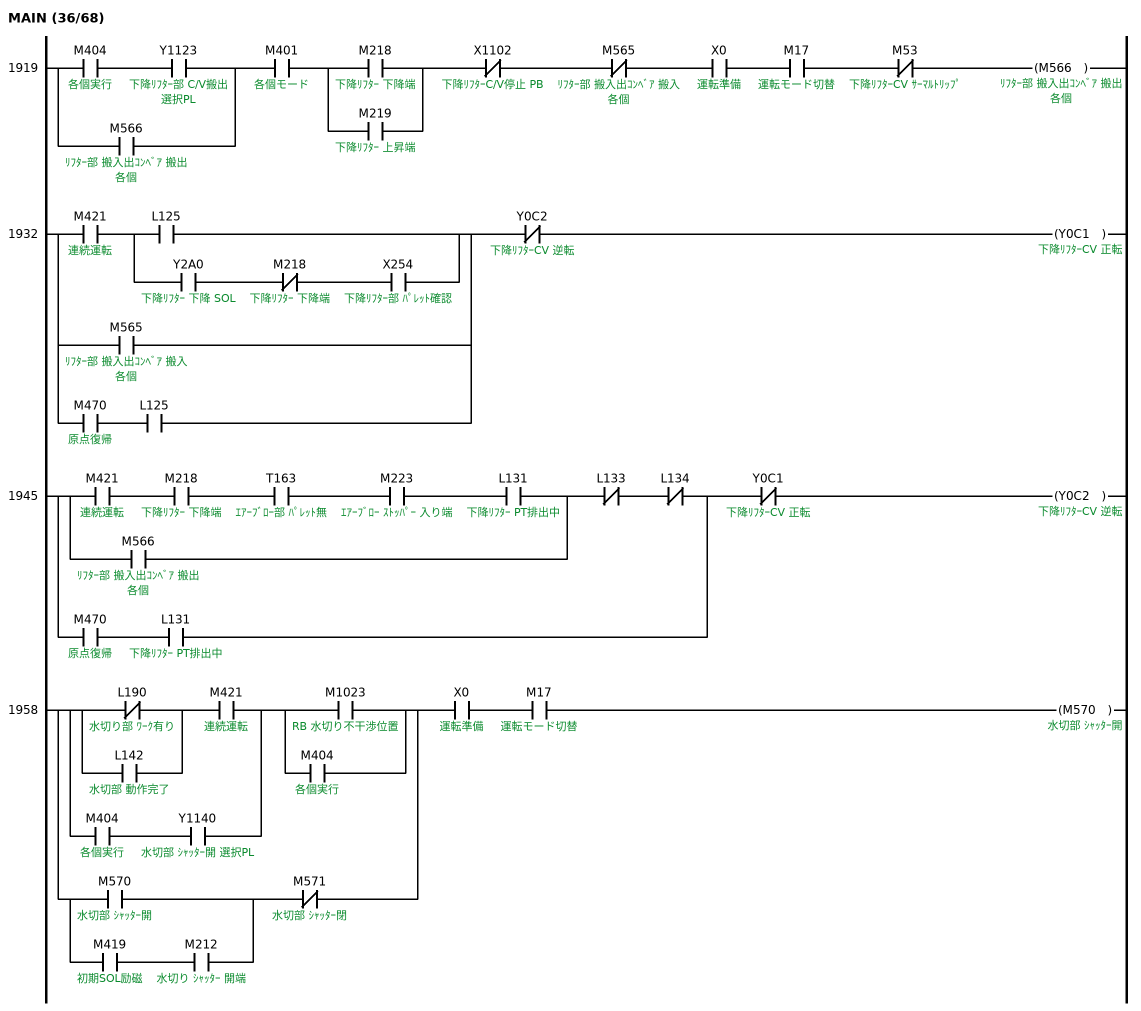
1919  LD      M404  ; 各個実行
      AND     Y1123  ; 下降ﾘﾌﾀｰ部 C/V搬出 選択PL
      OR      M566  ; ﾘﾌﾀｰ部 搬入出ｺﾝﾍﾞｱ 搬出 各個
      AND     M401  ; 各個モード
      LD      M218  ; 下降ﾘﾌﾀｰ 下降端
      OR      M219  ; 下降ﾘﾌﾀｰ 上昇端
      ANB
      ANI     X1102  ; 下降ﾘﾌﾀｰC/V停止 PB
      ANI     M565  ; ﾘﾌﾀｰ部 搬入出ｺﾝﾍﾞｱ 搬入 各個
      AND     X0  ; 運転準備
      AND     M17  ; 運転モード切替
      ANI     M53  ; 下降ﾘﾌﾀｰCV ｻｰﾏﾙﾄﾘｯﾌﾟ
      OUT     M566  ; ﾘﾌﾀｰ部 搬入出ｺﾝﾍﾞｱ 搬出 各個
1932  LD      M421  ; 連続運転
      LD      L125
      LD      Y2A0  ; 下降ﾘﾌﾀｰ 下降 SOL
      ANI     M218  ; 下降ﾘﾌﾀｰ 下降端
      AND     X254  ; 下降ﾘﾌﾀｰ部 ﾊﾟﾚｯﾄ確認
      ORB
      ANB
      OR      M565  ; ﾘﾌﾀｰ部 搬入出ｺﾝﾍﾞｱ 搬入 各個
      LD      M470  ; 原点復帰
      AND     L125
      ORB
      ANI     Y0C2  ; 下降ﾘﾌﾀｰCV 逆転
      OUT     Y0C1  ; 下降ﾘﾌﾀｰCV 正転
1945  LD      M421  ; 連続運転
      AND     M218  ; 下降ﾘﾌﾀｰ 下降端
      AND     T163  ; ｴｱｰﾌﾞﾛｰ部 ﾊﾟﾚｯﾄ無
      AND     M223  ; ｴｱｰﾌﾞﾛｰ ｽﾄｯﾊﾟｰ 入り端
      AND     L131  ; 下降ﾘﾌﾀｰ PT排出中
      OR      M566  ; ﾘﾌﾀｰ部 搬入出ｺﾝﾍﾞｱ 搬出 各個
      ANI     L133
      ANI     L134
      LD      M470  ; 原点復帰
      AND     L131  ; 下降ﾘﾌﾀｰ PT排出中
      ORB
      ANI     Y0C1  ; 下降ﾘﾌﾀｰCV 正転
      OUT     Y0C2  ; 下降ﾘﾌﾀｰCV 逆転
1958  LDI     L190  ; 水切り部 ﾜｰｸ有り
      OR      L142  ; 水切部 動作完了
      AND     M421  ; 連続運転
      LD      M404  ; 各個実行
      AND     Y1140  ; 水切部 ｼｬｯﾀｰ開 選択PL
      ORB
      LD      M1023  ; RB 水切り不干渉位置
      OR      M404  ; 各個実行
      ANB
      LD      M570  ; 水切部 ｼｬｯﾀｰ開
      LD      M419  ; 初期SOL励磁
      AND     M212  ; 水切り ｼｬｯﾀｰ 開端
      ORB
      ANI     M571  ; 水切部 ｼｬｯﾀｰ閉
      ORB
      AND     X0  ; 運転準備
      AND     M17  ; 運転モード切替
      OUT     M570  ; 水切部 ｼｬｯﾀｰ開
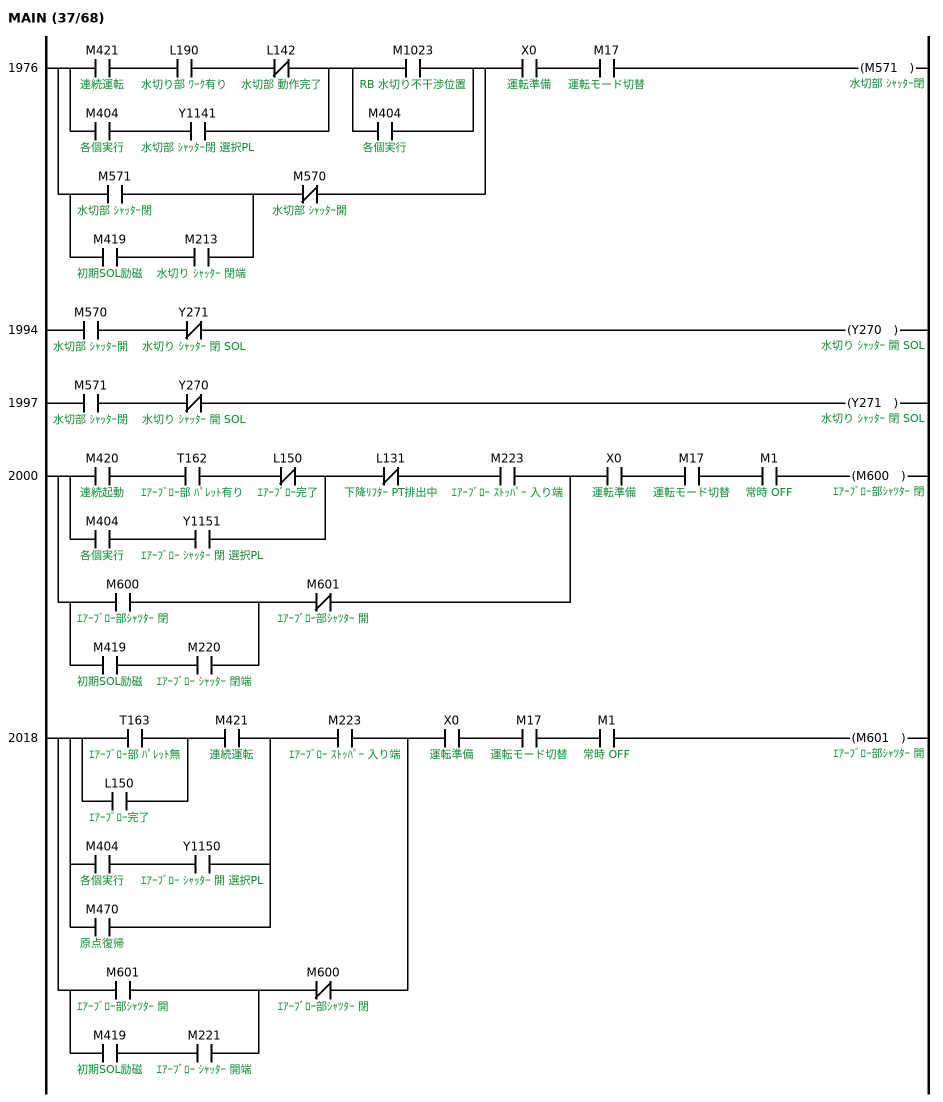
1976  LD      M421  ; 連続運転
      AND     L190  ; 水切り部 ﾜｰｸ有り
      ANI     L142  ; 水切部 動作完了
      LD      M404  ; 各個実行
      AND     Y1141  ; 水切部 ｼｬｯﾀｰ閉 選択PL
      ORB
      LD      M1023  ; RB 水切り不干渉位置
      OR      M404  ; 各個実行
      ANB
      LD      M571  ; 水切部 ｼｬｯﾀｰ閉
      LD      M419  ; 初期SOL励磁
      AND     M213  ; 水切り ｼｬｯﾀｰ 閉端
      ORB
      ANI     M570  ; 水切部 ｼｬｯﾀｰ開
      ORB
      AND     X0  ; 運転準備
      AND     M17  ; 運転モード切替
      OUT     M571  ; 水切部 ｼｬｯﾀｰ閉
1994  LD      M570  ; 水切部 ｼｬｯﾀｰ開
      ANI     Y271  ; 水切り ｼｬｯﾀｰ 閉 SOL
      OUT     Y270  ; 水切り ｼｬｯﾀｰ 開 SOL
1997  LD      M571  ; 水切部 ｼｬｯﾀｰ閉
      ANI     Y270  ; 水切り ｼｬｯﾀｰ 開 SOL
      OUT     Y271  ; 水切り ｼｬｯﾀｰ 閉 SOL
2000  LD      M420  ; 連続起動
      AND     T162  ; ｴｱｰﾌﾞﾛｰ部 ﾊﾟﾚｯﾄ有り
      ANI     L150  ; ｴｱｰﾌﾞﾛｰ完了
      LD      M404  ; 各個実行
      AND     Y1151  ; ｴｱｰﾌﾞﾛｰ ｼｬｯﾀｰ 閉 選択PL
      ORB
      ANI     L131  ; 下降ﾘﾌﾀｰ PT排出中
      AND     M223  ; ｴｱｰﾌﾞﾛｰ ｽﾄｯﾊﾟｰ 入り端
      LD      M600  ; ｴｱｰﾌﾞﾛｰ部ｼｬﾂﾀｰ 閉
      LD      M419  ; 初期SOL励磁
      AND     M220  ; ｴｱｰﾌﾞﾛｰ ｼｬｯﾀｰ 閉端
      ORB
      ANI     M601  ; ｴｱｰﾌﾞﾛｰ部ｼｬﾂﾀｰ 開
      ORB
      AND     X0  ; 運転準備
      AND     M17  ; 運転モード切替
      AND     M1  ; 常時 OFF
      OUT     M600  ; ｴｱｰﾌﾞﾛｰ部ｼｬﾂﾀｰ 閉
2018  LD      T163  ; ｴｱｰﾌﾞﾛｰ部 ﾊﾟﾚｯﾄ無
      OR      L150  ; ｴｱｰﾌﾞﾛｰ完了
      AND     M421  ; 連続運転
      LD      M404  ; 各個実行
      AND     Y1150  ; ｴｱｰﾌﾞﾛｰ ｼｬｯﾀｰ 開 選択PL
      ORB
      OR      M470  ; 原点復帰
      AND     M223  ; ｴｱｰﾌﾞﾛｰ ｽﾄｯﾊﾟｰ 入り端
      LD      M601  ; ｴｱｰﾌﾞﾛｰ部ｼｬﾂﾀｰ 開
      LD      M419  ; 初期SOL励磁
      AND     M221  ; ｴｱｰﾌﾞﾛｰ ｼｬｯﾀｰ 開端
      ORB
      ANI     M600  ; ｴｱｰﾌﾞﾛｰ部ｼｬﾂﾀｰ 閉
      ORB
      AND     X0  ; 運転準備
      AND     M17  ; 運転モード切替
      AND     M1  ; 常時 OFF
      OUT     M601  ; ｴｱｰﾌﾞﾛｰ部ｼｬﾂﾀｰ 開
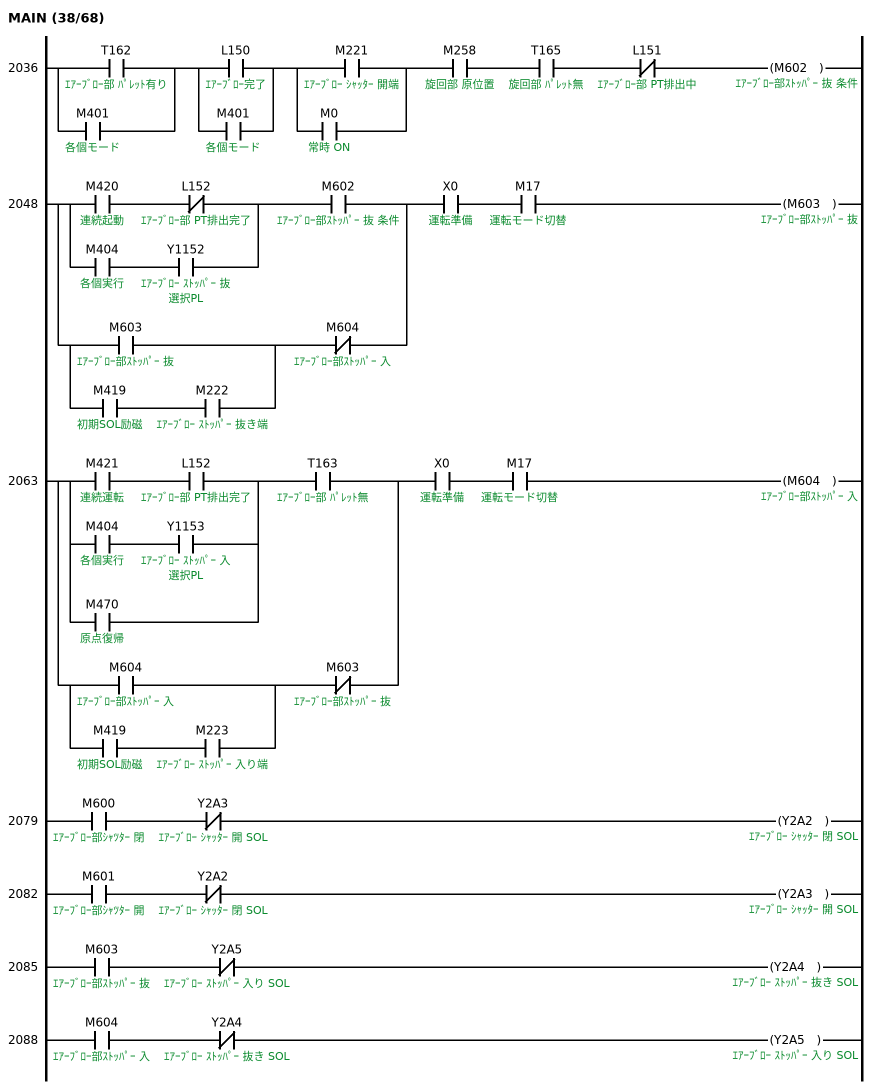
2036  LD      T162  ; ｴｱｰﾌﾞﾛｰ部 ﾊﾟﾚｯﾄ有り
      OR      M401  ; 各個モード
      LD      L150  ; ｴｱｰﾌﾞﾛｰ完了
      OR      M401  ; 各個モード
      ANB
      LD      M221  ; ｴｱｰﾌﾞﾛｰ ｼｬｯﾀｰ 開端
      OR      M0  ; 常時 ON
      ANB
      AND     M258  ; 旋回部 原位置
      AND     T165  ; 旋回部 ﾊﾟﾚｯﾄ無
      ANI     L151  ; ｴｱｰﾌﾞﾛｰ部 PT排出中
      OUT     M602  ; ｴｱｰﾌﾞﾛｰ部ｽﾄｯﾊﾟｰ 抜 条件
2048  LD      M420  ; 連続起動
      ANI     L152  ; ｴｱｰﾌﾞﾛｰ部 PT排出完了
      LD      M404  ; 各個実行
      AND     Y1152  ; ｴｱｰﾌﾞﾛｰ ｽﾄｯﾊﾟｰ 抜 選択PL
      ORB
      AND     M602  ; ｴｱｰﾌﾞﾛｰ部ｽﾄｯﾊﾟｰ 抜 条件
      LD      M603  ; ｴｱｰﾌﾞﾛｰ部ｽﾄｯﾊﾟｰ 抜
      LD      M419  ; 初期SOL励磁
      AND     M222  ; ｴｱｰﾌﾞﾛｰ ｽﾄｯﾊﾟｰ 抜き端
      ORB
      ANI     M604  ; ｴｱｰﾌﾞﾛｰ部ｽﾄｯﾊﾟｰ 入
      ORB
      AND     X0  ; 運転準備
      AND     M17  ; 運転モード切替
      OUT     M603  ; ｴｱｰﾌﾞﾛｰ部ｽﾄｯﾊﾟｰ 抜
2063  LD      M421  ; 連続運転
      AND     L152  ; ｴｱｰﾌﾞﾛｰ部 PT排出完了
      LD      M404  ; 各個実行
      AND     Y1153  ; ｴｱｰﾌﾞﾛｰ ｽﾄｯﾊﾟｰ 入 選択PL
      ORB
      OR      M470  ; 原点復帰
      AND     T163  ; ｴｱｰﾌﾞﾛｰ部 ﾊﾟﾚｯﾄ無
      LD      M604  ; ｴｱｰﾌﾞﾛｰ部ｽﾄｯﾊﾟｰ 入
      LD      M419  ; 初期SOL励磁
      AND     M223  ; ｴｱｰﾌﾞﾛｰ ｽﾄｯﾊﾟｰ 入り端
      ORB
      ANI     M603  ; ｴｱｰﾌﾞﾛｰ部ｽﾄｯﾊﾟｰ 抜
      ORB
      AND     X0  ; 運転準備
      AND     M17  ; 運転モード切替
      OUT     M604  ; ｴｱｰﾌﾞﾛｰ部ｽﾄｯﾊﾟｰ 入
2079  LD      M600  ; ｴｱｰﾌﾞﾛｰ部ｼｬﾂﾀｰ 閉
      ANI     Y2A3  ; ｴｱｰﾌﾞﾛｰ ｼｬｯﾀｰ 開 SOL
      OUT     Y2A2  ; ｴｱｰﾌﾞﾛｰ ｼｬｯﾀｰ 閉 SOL
2082  LD      M601  ; ｴｱｰﾌﾞﾛｰ部ｼｬﾂﾀｰ 開
      ANI     Y2A2  ; ｴｱｰﾌﾞﾛｰ ｼｬｯﾀｰ 閉 SOL
      OUT     Y2A3  ; ｴｱｰﾌﾞﾛｰ ｼｬｯﾀｰ 開 SOL
2085  LD      M603  ; ｴｱｰﾌﾞﾛｰ部ｽﾄｯﾊﾟｰ 抜
      ANI     Y2A5  ; ｴｱｰﾌﾞﾛｰ ｽﾄｯﾊﾟｰ 入り SOL
      OUT     Y2A4  ; ｴｱｰﾌﾞﾛｰ ｽﾄｯﾊﾟｰ 抜き SOL
2088  LD      M604  ; ｴｱｰﾌﾞﾛｰ部ｽﾄｯﾊﾟｰ 入
      ANI     Y2A4  ; ｴｱｰﾌﾞﾛｰ ｽﾄｯﾊﾟｰ 抜き SOL
      OUT     Y2A5  ; ｴｱｰﾌﾞﾛｰ ｽﾄｯﾊﾟｰ 入り SOL
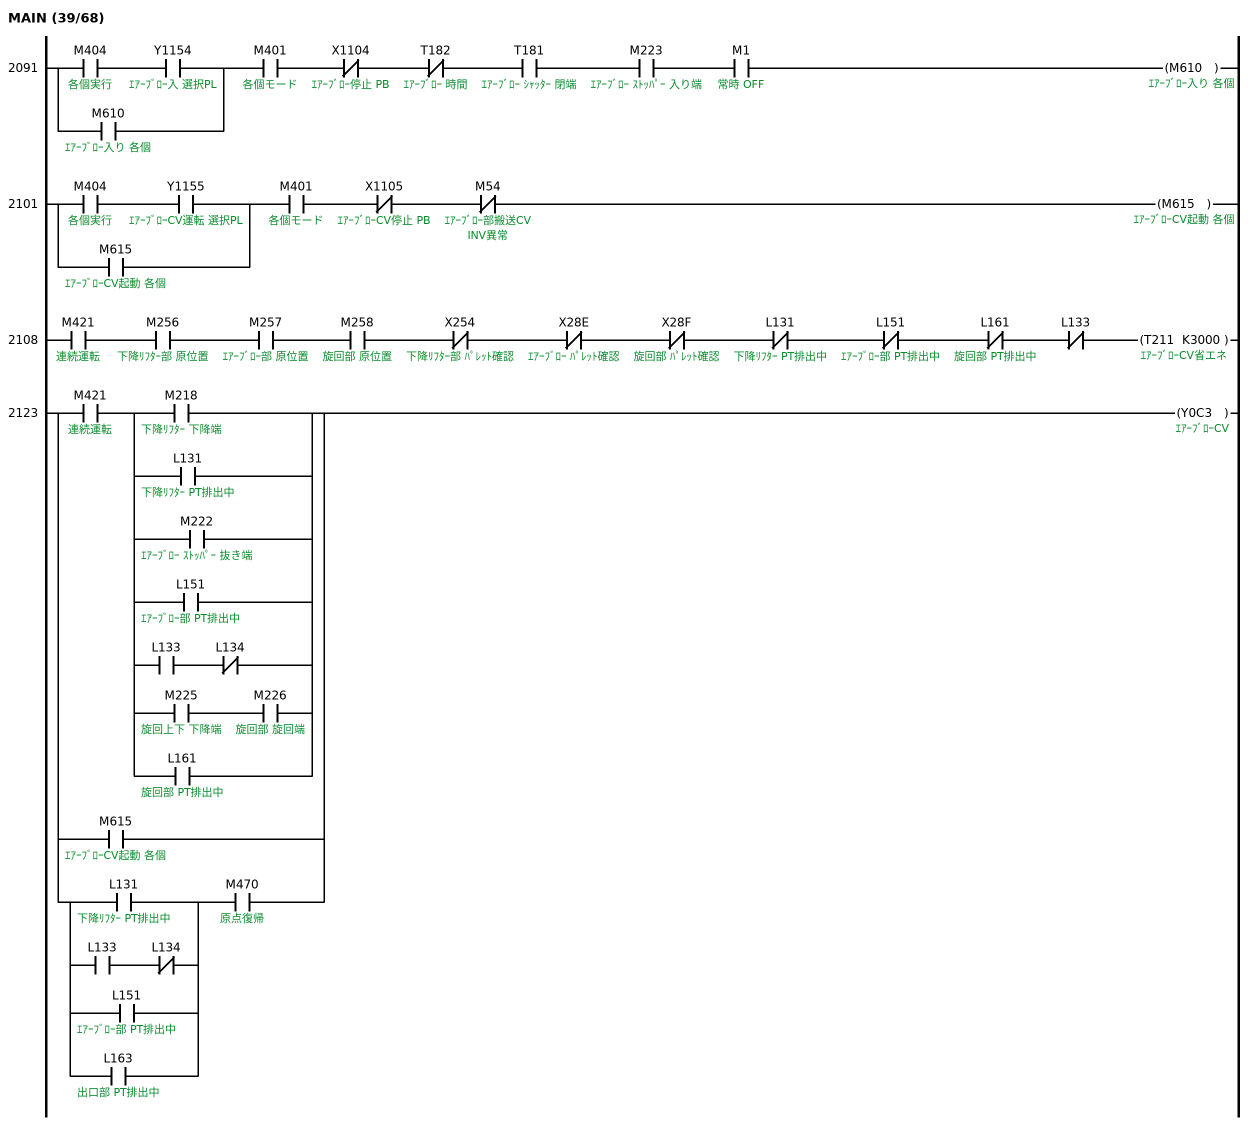
2091  LD      M404  ; 各個実行
      AND     Y1154  ; ｴｱｰﾌﾞﾛｰ入 選択PL
      OR      M610  ; ｴｱｰﾌﾞﾛｰ入り 各個
      AND     M401  ; 各個モード
      ANI     X1104  ; ｴｱｰﾌﾞﾛｰ停止 PB
      ANI     T182  ; ｴｱｰﾌﾞﾛｰ 時間
      AND     T181  ; ｴｱｰﾌﾞﾛｰ ｼｬｯﾀｰ 閉端
      AND     M223  ; ｴｱｰﾌﾞﾛｰ ｽﾄｯﾊﾟｰ 入り端
      AND     M1  ; 常時 OFF
      OUT     M610  ; ｴｱｰﾌﾞﾛｰ入り 各個
2101  LD      M404  ; 各個実行
      AND     Y1155  ; ｴｱｰﾌﾞﾛｰCV運転 選択PL
      OR      M615  ; ｴｱｰﾌﾞﾛｰCV起動 各個
      AND     M401  ; 各個モード
      ANI     X1105  ; ｴｱｰﾌﾞﾛｰCV停止 PB
      ANI     M54  ; ｴｱｰﾌﾞﾛｰ部搬送CV INV異常
      OUT     M615  ; ｴｱｰﾌﾞﾛｰCV起動 各個
2108  LD      M421  ; 連続運転
      AND     M256  ; 下降ﾘﾌﾀｰ部 原位置
      AND     M257  ; ｴｱｰﾌﾞﾛｰ部 原位置
      AND     M258  ; 旋回部 原位置
      ANI     X254  ; 下降ﾘﾌﾀｰ部 ﾊﾟﾚｯﾄ確認
      ANI     X28E  ; ｴｱｰﾌﾞﾛｰ ﾊﾟﾚｯﾄ確認
      ANI     X28F  ; 旋回部 ﾊﾟﾚｯﾄ確認
      ANI     L131  ; 下降ﾘﾌﾀｰ PT排出中
      ANI     L151  ; ｴｱｰﾌﾞﾛｰ部 PT排出中
      ANI     L161  ; 旋回部 PT排出中
      ANI     L133
      OUT     T211 K3000  ; ｴｱｰﾌﾞﾛｰCV省エネ
2123  LD      M421  ; 連続運転
      LD      M218  ; 下降ﾘﾌﾀｰ 下降端
      OR      L131  ; 下降ﾘﾌﾀｰ PT排出中
      OR      M222  ; ｴｱｰﾌﾞﾛｰ ｽﾄｯﾊﾟｰ 抜き端
      OR      L151  ; ｴｱｰﾌﾞﾛｰ部 PT排出中
      LD      L133
      ANI     L134
      ORB
      LD      M225  ; 旋回上下 下降端
      AND     M226  ; 旋回部 旋回端
      ORB
      OR      L161  ; 旋回部 PT排出中
      ANB
      OR      M615  ; ｴｱｰﾌﾞﾛｰCV起動 各個
      LD      L131  ; 下降ﾘﾌﾀｰ PT排出中
      LD      L133
      ANI     L134
      ORB
      OR      L151  ; ｴｱｰﾌﾞﾛｰ部 PT排出中
      OR      L163  ; 出口部 PT排出中
      AND     M470  ; 原点復帰
      ORB
      OUT     Y0C3  ; ｴｱｰﾌﾞﾛｰCV
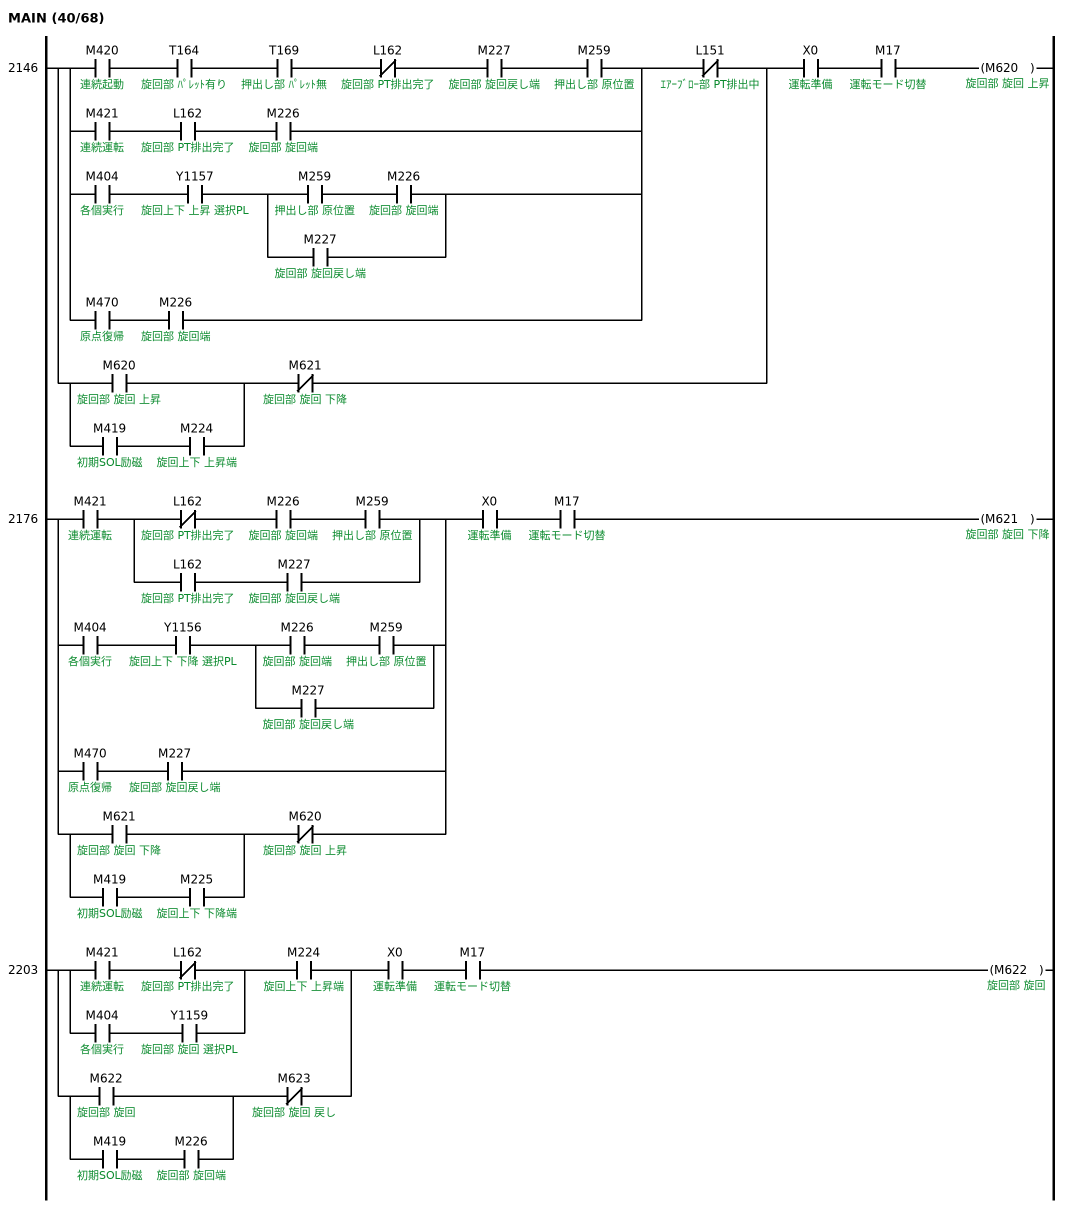
2146  LD      M420  ; 連続起動
      AND     T164  ; 旋回部 ﾊﾟﾚｯﾄ有り
      AND     T169  ; 押出し部 ﾊﾟﾚｯﾄ無
      ANI     L162  ; 旋回部 PT排出完了
      AND     M227  ; 旋回部 旋回戻し端
      AND     M259  ; 押出し部 原位置
      LD      M421  ; 連続運転
      AND     L162  ; 旋回部 PT排出完了
      AND     M226  ; 旋回部 旋回端
      ORB
      LD      M404  ; 各個実行
      AND     Y1157  ; 旋回上下 上昇 選択PL
      LD      M259  ; 押出し部 原位置
      AND     M226  ; 旋回部 旋回端
      OR      M227  ; 旋回部 旋回戻し端
      ANB
      ORB
      LD      M470  ; 原点復帰
      AND     M226  ; 旋回部 旋回端
      ORB
      ANI     L151  ; ｴｱｰﾌﾞﾛｰ部 PT排出中
      LD      M620  ; 旋回部 旋回 上昇
      LD      M419  ; 初期SOL励磁
      AND     M224  ; 旋回上下 上昇端
      ORB
      ANI     M621  ; 旋回部 旋回 下降
      ORB
      AND     X0  ; 運転準備
      AND     M17  ; 運転モード切替
      OUT     M620  ; 旋回部 旋回 上昇
2176  LD      M421  ; 連続運転
      LDI     L162  ; 旋回部 PT排出完了
      AND     M226  ; 旋回部 旋回端
      AND     M259  ; 押出し部 原位置
      LD      L162  ; 旋回部 PT排出完了
      AND     M227  ; 旋回部 旋回戻し端
      ORB
      ANB
      LD      M404  ; 各個実行
      AND     Y1156  ; 旋回上下 下降 選択PL
      LD      M226  ; 旋回部 旋回端
      AND     M259  ; 押出し部 原位置
      OR      M227  ; 旋回部 旋回戻し端
      ANB
      ORB
      LD      M470  ; 原点復帰
      AND     M227  ; 旋回部 旋回戻し端
      ORB
      LD      M621  ; 旋回部 旋回 下降
      LD      M419  ; 初期SOL励磁
      AND     M225  ; 旋回上下 下降端
      ORB
      ANI     M620  ; 旋回部 旋回 上昇
      ORB
      AND     X0  ; 運転準備
      AND     M17  ; 運転モード切替
      OUT     M621  ; 旋回部 旋回 下降
2203  LD      M421  ; 連続運転
      ANI     L162  ; 旋回部 PT排出完了
      LD      M404  ; 各個実行
      AND     Y1159  ; 旋回部 旋回 選択PL
      ORB
      AND     M224  ; 旋回上下 上昇端
      LD      M622  ; 旋回部 旋回
      LD      M419  ; 初期SOL励磁
      AND     M226  ; 旋回部 旋回端
      ORB
      ANI     M623  ; 旋回部 旋回 戻し
      ORB
      AND     X0  ; 運転準備
      AND     M17  ; 運転モード切替
      OUT     M622  ; 旋回部 旋回
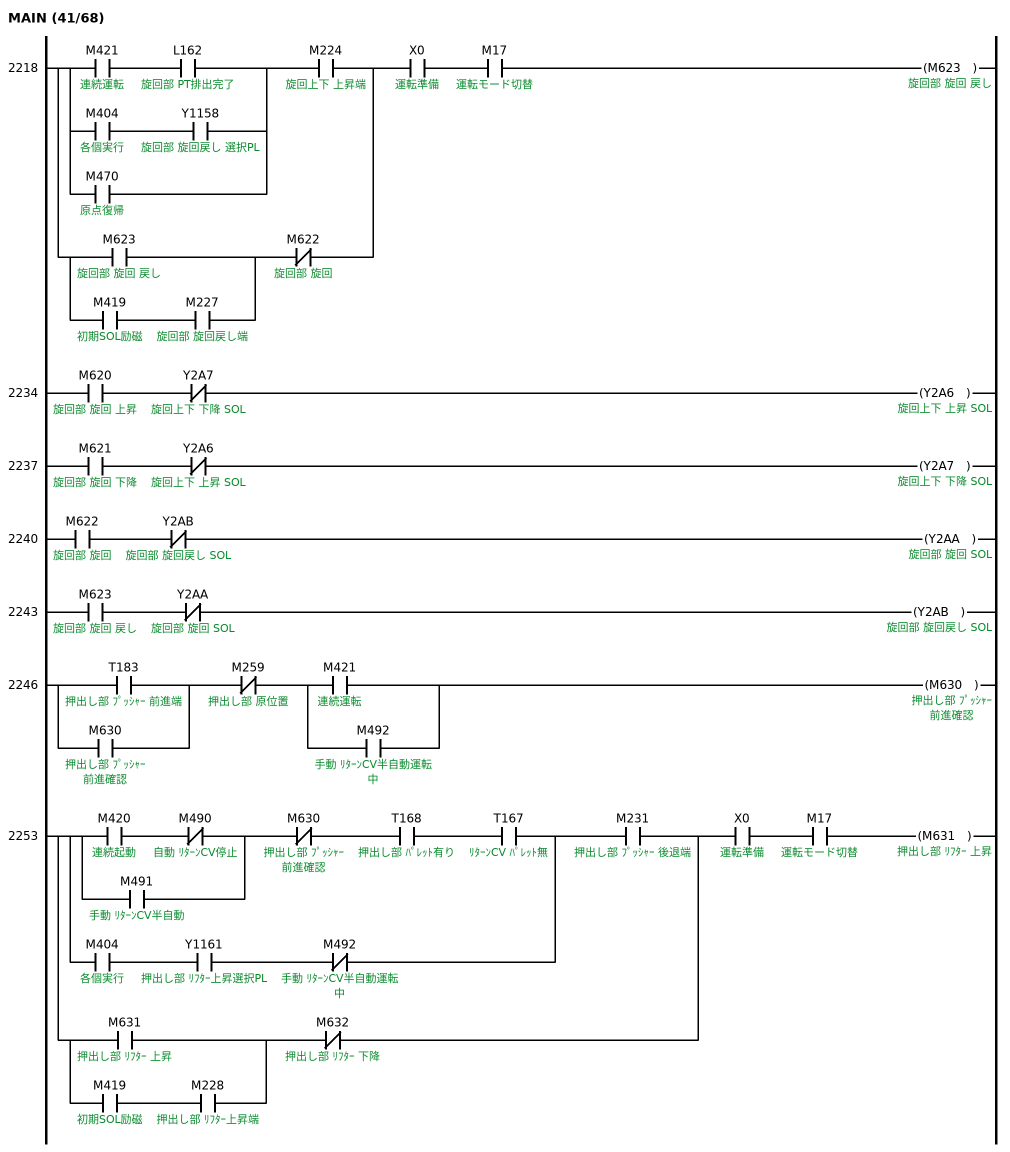
2218  LD      M421  ; 連続運転
      AND     L162  ; 旋回部 PT排出完了
      LD      M404  ; 各個実行
      AND     Y1158  ; 旋回部 旋回戻し 選択PL
      ORB
      OR      M470  ; 原点復帰
      AND     M224  ; 旋回上下 上昇端
      LD      M623  ; 旋回部 旋回 戻し
      LD      M419  ; 初期SOL励磁
      AND     M227  ; 旋回部 旋回戻し端
      ORB
      ANI     M622  ; 旋回部 旋回
      ORB
      AND     X0  ; 運転準備
      AND     M17  ; 運転モード切替
      OUT     M623  ; 旋回部 旋回 戻し
2234  LD      M620  ; 旋回部 旋回 上昇
      ANI     Y2A7  ; 旋回上下 下降 SOL
      OUT     Y2A6  ; 旋回上下 上昇 SOL
2237  LD      M621  ; 旋回部 旋回 下降
      ANI     Y2A6  ; 旋回上下 上昇 SOL
      OUT     Y2A7  ; 旋回上下 下降 SOL
2240  LD      M622  ; 旋回部 旋回
      ANI     Y2AB  ; 旋回部 旋回戻し SOL
      OUT     Y2AA  ; 旋回部 旋回 SOL
2243  LD      M623  ; 旋回部 旋回 戻し
      ANI     Y2AA  ; 旋回部 旋回 SOL
      OUT     Y2AB  ; 旋回部 旋回戻し SOL
2246  LD      T183  ; 押出し部 ﾌﾟｯｼｬｰ 前進端
      OR      M630  ; 押出し部 ﾌﾟｯｼｬｰ 前進確認
      ANI     M259  ; 押出し部 原位置
      LD      M421  ; 連続運転
      OR      M492  ; 手動 ﾘﾀｰﾝCV半自動運転中
      ANB
      OUT     M630  ; 押出し部 ﾌﾟｯｼｬｰ 前進確認
2253  LD      M420  ; 連続起動
      ANI     M490  ; 自動 ﾘﾀｰﾝCV停止
      OR      M491  ; 手動 ﾘﾀｰﾝCV半自動
      ANI     M630  ; 押出し部 ﾌﾟｯｼｬｰ 前進確認
      AND     T168  ; 押出し部 ﾊﾟﾚｯﾄ有り
      AND     T167  ; ﾘﾀｰﾝCV ﾊﾟﾚｯﾄ無
      LD      M404  ; 各個実行
      AND     Y1161  ; 押出し部 ﾘﾌﾀｰ上昇選択PL
      ANI     M492  ; 手動 ﾘﾀｰﾝCV半自動運転中
      ORB
      AND     M231  ; 押出し部 ﾌﾟｯｼｬｰ 後退端
      LD      M631  ; 押出し部 ﾘﾌﾀｰ 上昇
      LD      M419  ; 初期SOL励磁
      AND     M228  ; 押出し部 ﾘﾌﾀｰ上昇端
      ORB
      ANI     M632  ; 押出し部 ﾘﾌﾀｰ 下降
      ORB
      AND     X0  ; 運転準備
      AND     M17  ; 運転モード切替
      OUT     M631  ; 押出し部 ﾘﾌﾀｰ 上昇
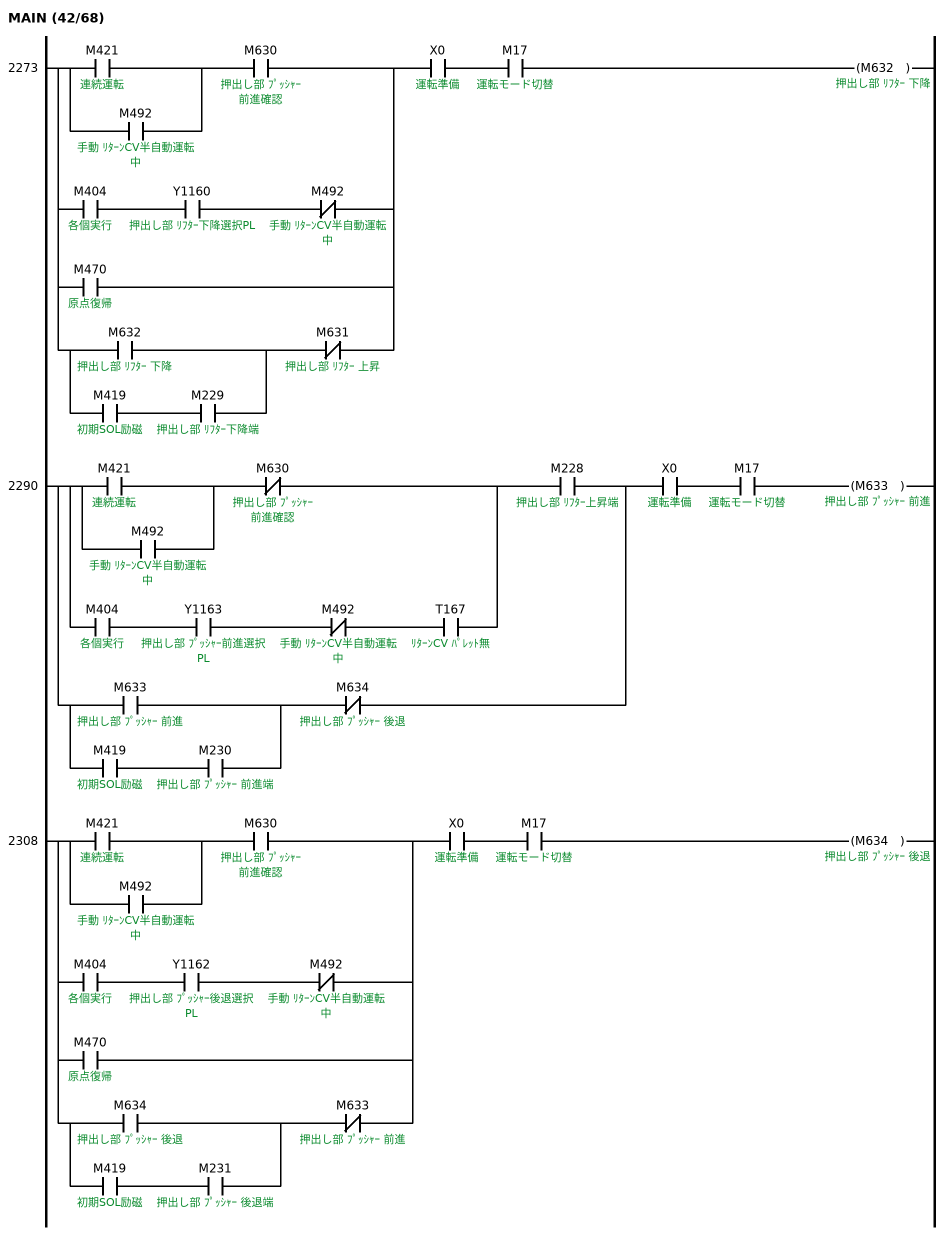
2273  LD      M421  ; 連続運転
      OR      M492  ; 手動 ﾘﾀｰﾝCV半自動運転中
      AND     M630  ; 押出し部 ﾌﾟｯｼｬｰ 前進確認
      LD      M404  ; 各個実行
      AND     Y1160  ; 押出し部 ﾘﾌﾀｰ下降選択PL
      ANI     M492  ; 手動 ﾘﾀｰﾝCV半自動運転中
      ORB
      OR      M470  ; 原点復帰
      LD      M632  ; 押出し部 ﾘﾌﾀｰ 下降
      LD      M419  ; 初期SOL励磁
      AND     M229  ; 押出し部 ﾘﾌﾀｰ下降端
      ORB
      ANI     M631  ; 押出し部 ﾘﾌﾀｰ 上昇
      ORB
      AND     X0  ; 運転準備
      AND     M17  ; 運転モード切替
      OUT     M632  ; 押出し部 ﾘﾌﾀｰ 下降
2290  LD      M421  ; 連続運転
      OR      M492  ; 手動 ﾘﾀｰﾝCV半自動運転中
      ANI     M630  ; 押出し部 ﾌﾟｯｼｬｰ 前進確認
      LD      M404  ; 各個実行
      AND     Y1163  ; 押出し部 ﾌﾟｯｼｬｰ前進選択PL
      ANI     M492  ; 手動 ﾘﾀｰﾝCV半自動運転中
      AND     T167  ; ﾘﾀｰﾝCV ﾊﾟﾚｯﾄ無
      ORB
      AND     M228  ; 押出し部 ﾘﾌﾀｰ上昇端
      LD      M633  ; 押出し部 ﾌﾟｯｼｬｰ 前進
      LD      M419  ; 初期SOL励磁
      AND     M230  ; 押出し部 ﾌﾟｯｼｬｰ 前進端
      ORB
      ANI     M634  ; 押出し部 ﾌﾟｯｼｬｰ 後退
      ORB
      AND     X0  ; 運転準備
      AND     M17  ; 運転モード切替
      OUT     M633  ; 押出し部 ﾌﾟｯｼｬｰ 前進
2308  LD      M421  ; 連続運転
      OR      M492  ; 手動 ﾘﾀｰﾝCV半自動運転中
      AND     M630  ; 押出し部 ﾌﾟｯｼｬｰ 前進確認
      LD      M404  ; 各個実行
      AND     Y1162  ; 押出し部 ﾌﾟｯｼｬｰ後退選択PL
      ANI     M492  ; 手動 ﾘﾀｰﾝCV半自動運転中
      ORB
      OR      M470  ; 原点復帰
      LD      M634  ; 押出し部 ﾌﾟｯｼｬｰ 後退
      LD      M419  ; 初期SOL励磁
      AND     M231  ; 押出し部 ﾌﾟｯｼｬｰ 後退端
      ORB
      ANI     M633  ; 押出し部 ﾌﾟｯｼｬｰ 前進
      ORB
      AND     X0  ; 運転準備
      AND     M17  ; 運転モード切替
      OUT     M634  ; 押出し部 ﾌﾟｯｼｬｰ 後退
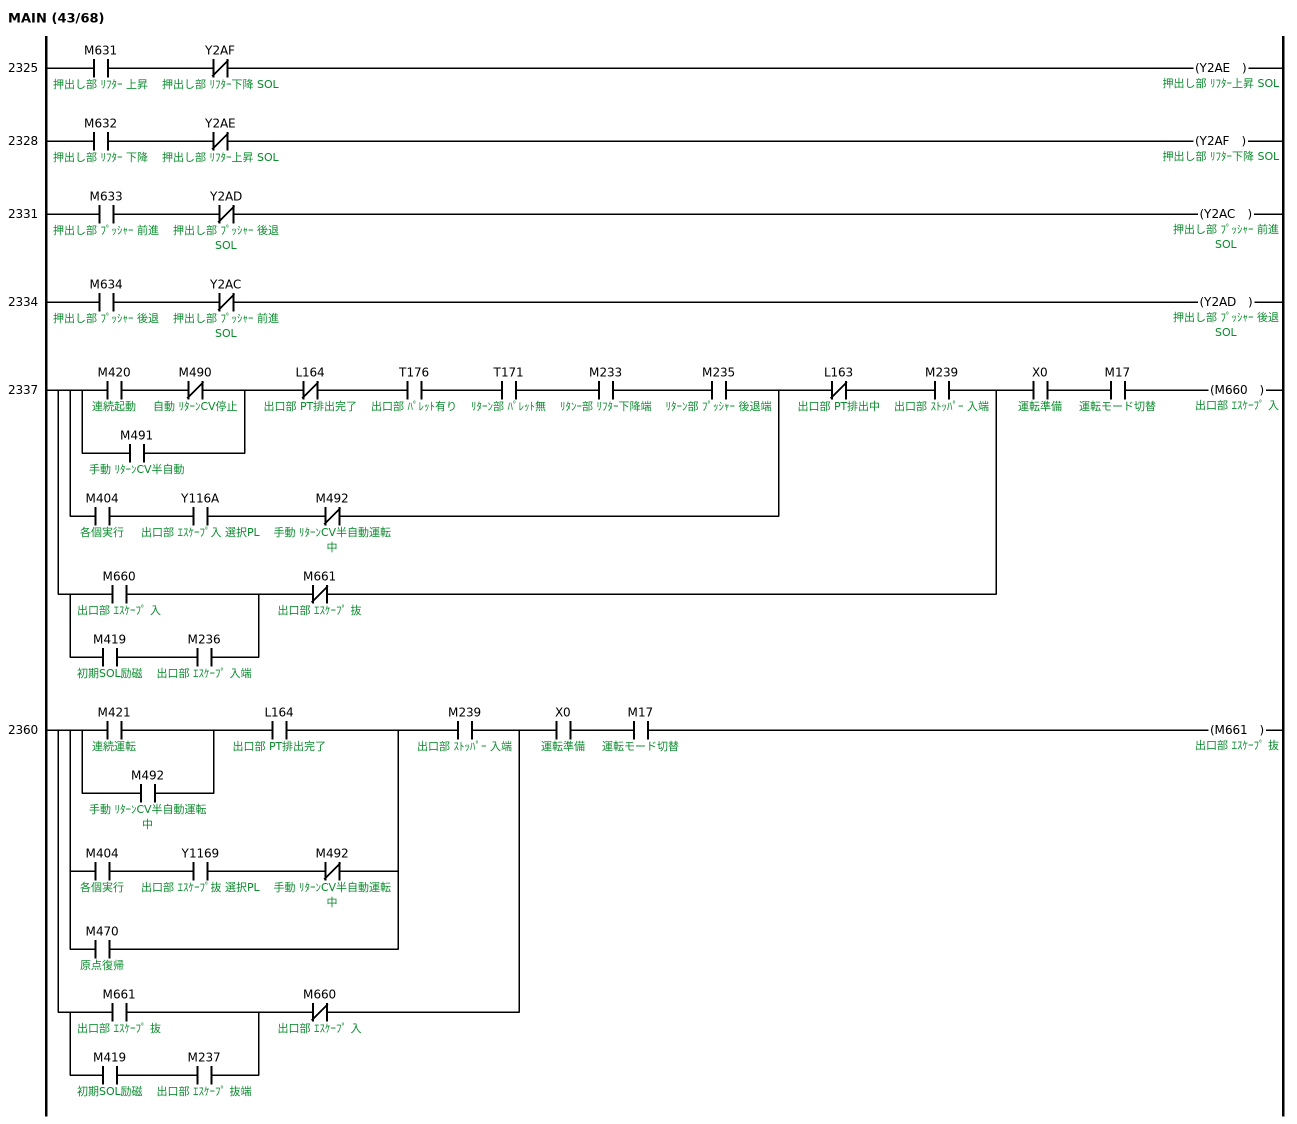
2325  LD      M631  ; 押出し部 ﾘﾌﾀｰ 上昇
      ANI     Y2AF  ; 押出し部 ﾘﾌﾀｰ下降 SOL
      OUT     Y2AE  ; 押出し部 ﾘﾌﾀｰ上昇 SOL
2328  LD      M632  ; 押出し部 ﾘﾌﾀｰ 下降
      ANI     Y2AE  ; 押出し部 ﾘﾌﾀｰ上昇 SOL
      OUT     Y2AF  ; 押出し部 ﾘﾌﾀｰ下降 SOL
2331  LD      M633  ; 押出し部 ﾌﾟｯｼｬｰ 前進
      ANI     Y2AD  ; 押出し部 ﾌﾟｯｼｬｰ 後退 SOL
      OUT     Y2AC  ; 押出し部 ﾌﾟｯｼｬｰ 前進 SOL
2334  LD      M634  ; 押出し部 ﾌﾟｯｼｬｰ 後退
      ANI     Y2AC  ; 押出し部 ﾌﾟｯｼｬｰ 前進 SOL
      OUT     Y2AD  ; 押出し部 ﾌﾟｯｼｬｰ 後退 SOL
2337  LD      M420  ; 連続起動
      ANI     M490  ; 自動 ﾘﾀｰﾝCV停止
      OR      M491  ; 手動 ﾘﾀｰﾝCV半自動
      ANI     L164  ; 出口部 PT排出完了
      AND     T176  ; 出口部 ﾊﾟﾚｯﾄ有り
      AND     T171  ; ﾘﾀｰﾝ部 ﾊﾟﾚｯﾄ無
      AND     M233  ; ﾘﾀﾝｰ部 ﾘﾌﾀｰ下降端
      AND     M235  ; ﾘﾀｰﾝ部 ﾌﾟｯｼｬｰ 後退端
      LD      M404  ; 各個実行
      AND     Y116A  ; 出口部 ｴｽｹｰﾌﾟ入 選択PL
      ANI     M492  ; 手動 ﾘﾀｰﾝCV半自動運転中
      ORB
      ANI     L163  ; 出口部 PT排出中
      AND     M239  ; 出口部 ｽﾄｯﾊﾟｰ 入端
      LD      M660  ; 出口部 ｴｽｹｰﾌﾟ 入
      LD      M419  ; 初期SOL励磁
      AND     M236  ; 出口部 ｴｽｹｰﾌﾟ 入端
      ORB
      ANI     M661  ; 出口部 ｴｽｹｰﾌﾟ 抜
      ORB
      AND     X0  ; 運転準備
      AND     M17  ; 運転モード切替
      OUT     M660  ; 出口部 ｴｽｹｰﾌﾟ 入
2360  LD      M421  ; 連続運転
      OR      M492  ; 手動 ﾘﾀｰﾝCV半自動運転中
      AND     L164  ; 出口部 PT排出完了
      LD      M404  ; 各個実行
      AND     Y1169  ; 出口部 ｴｽｹｰﾌﾟ抜 選択PL
      ANI     M492  ; 手動 ﾘﾀｰﾝCV半自動運転中
      ORB
      OR      M470  ; 原点復帰
      AND     M239  ; 出口部 ｽﾄｯﾊﾟｰ 入端
      LD      M661  ; 出口部 ｴｽｹｰﾌﾟ 抜
      LD      M419  ; 初期SOL励磁
      AND     M237  ; 出口部 ｴｽｹｰﾌﾟ 抜端
      ORB
      ANI     M660  ; 出口部 ｴｽｹｰﾌﾟ 入
      ORB
      AND     X0  ; 運転準備
      AND     M17  ; 運転モード切替
      OUT     M661  ; 出口部 ｴｽｹｰﾌﾟ 抜
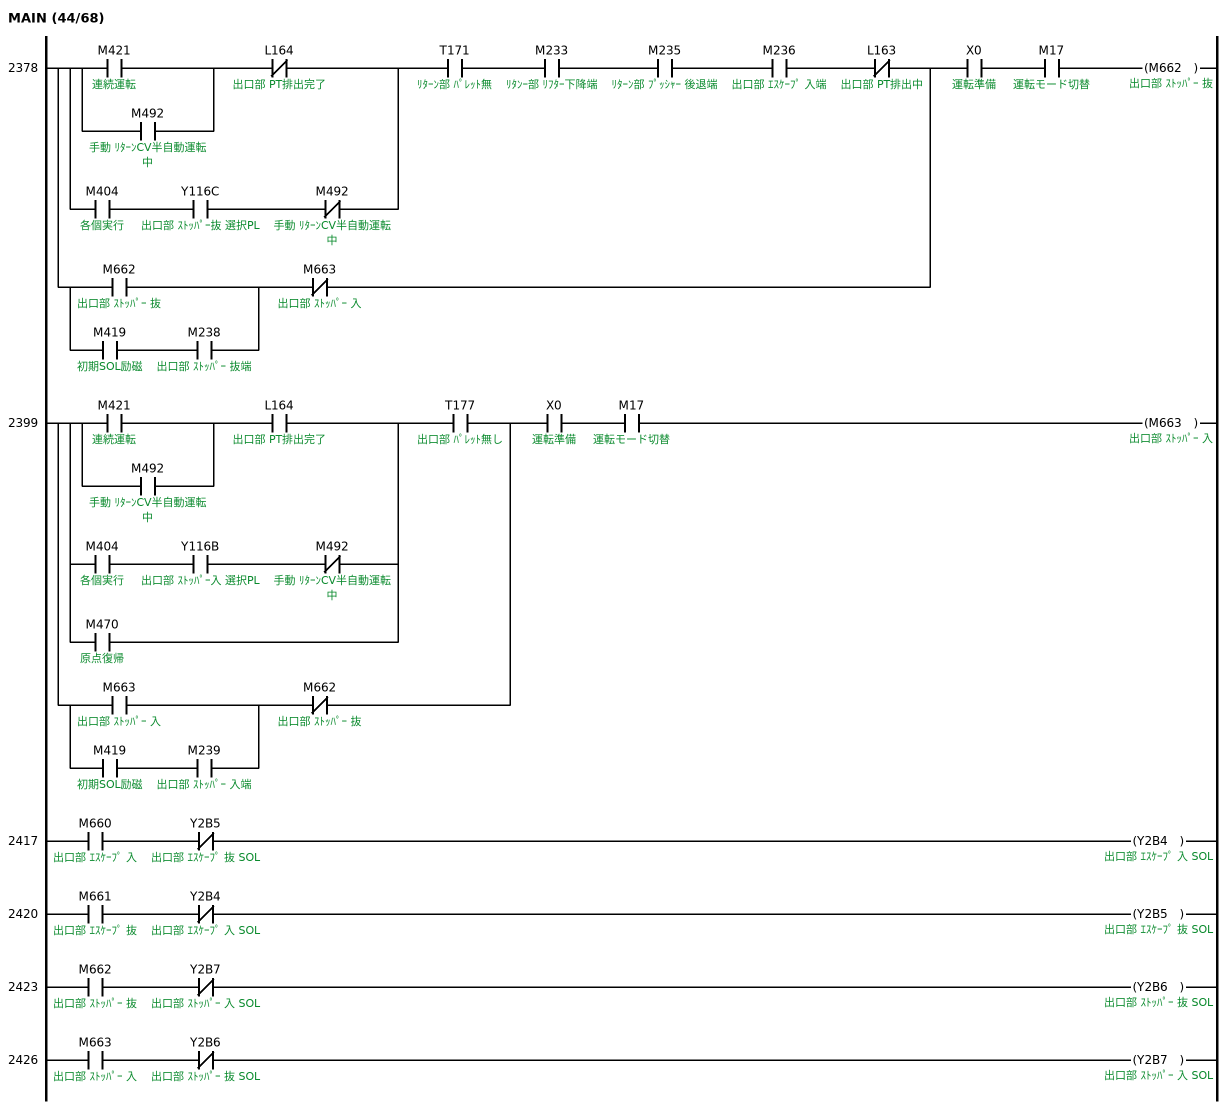
2378  LD      M421  ; 連続運転
      OR      M492  ; 手動 ﾘﾀｰﾝCV半自動運転中
      ANI     L164  ; 出口部 PT排出完了
      LD      M404  ; 各個実行
      AND     Y116C  ; 出口部 ｽﾄｯﾊﾟｰ抜 選択PL
      ANI     M492  ; 手動 ﾘﾀｰﾝCV半自動運転中
      ORB
      AND     T171  ; ﾘﾀｰﾝ部 ﾊﾟﾚｯﾄ無
      AND     M233  ; ﾘﾀﾝｰ部 ﾘﾌﾀｰ下降端
      AND     M235  ; ﾘﾀｰﾝ部 ﾌﾟｯｼｬｰ 後退端
      AND     M236  ; 出口部 ｴｽｹｰﾌﾟ 入端
      ANI     L163  ; 出口部 PT排出中
      LD      M662  ; 出口部 ｽﾄｯﾊﾟｰ 抜
      LD      M419  ; 初期SOL励磁
      AND     M238  ; 出口部 ｽﾄｯﾊﾟｰ 抜端
      ORB
      ANI     M663  ; 出口部 ｽﾄｯﾊﾟｰ 入
      ORB
      AND     X0  ; 運転準備
      AND     M17  ; 運転モード切替
      OUT     M662  ; 出口部 ｽﾄｯﾊﾟｰ 抜
2399  LD      M421  ; 連続運転
      OR      M492  ; 手動 ﾘﾀｰﾝCV半自動運転中
      AND     L164  ; 出口部 PT排出完了
      LD      M404  ; 各個実行
      AND     Y116B  ; 出口部 ｽﾄｯﾊﾟｰ入 選択PL
      ANI     M492  ; 手動 ﾘﾀｰﾝCV半自動運転中
      ORB
      OR      M470  ; 原点復帰
      AND     T177  ; 出口部 ﾊﾟﾚｯﾄ無し
      LD      M663  ; 出口部 ｽﾄｯﾊﾟｰ 入
      LD      M419  ; 初期SOL励磁
      AND     M239  ; 出口部 ｽﾄｯﾊﾟｰ 入端
      ORB
      ANI     M662  ; 出口部 ｽﾄｯﾊﾟｰ 抜
      ORB
      AND     X0  ; 運転準備
      AND     M17  ; 運転モード切替
      OUT     M663  ; 出口部 ｽﾄｯﾊﾟｰ 入
2417  LD      M660  ; 出口部 ｴｽｹｰﾌﾟ 入
      ANI     Y2B5  ; 出口部 ｴｽｹｰﾌﾟ 抜 SOL
      OUT     Y2B4  ; 出口部 ｴｽｹｰﾌﾟ 入 SOL
2420  LD      M661  ; 出口部 ｴｽｹｰﾌﾟ 抜
      ANI     Y2B4  ; 出口部 ｴｽｹｰﾌﾟ 入 SOL
      OUT     Y2B5  ; 出口部 ｴｽｹｰﾌﾟ 抜 SOL
2423  LD      M662  ; 出口部 ｽﾄｯﾊﾟｰ 抜
      ANI     Y2B7  ; 出口部 ｽﾄｯﾊﾟｰ 入 SOL
      OUT     Y2B6  ; 出口部 ｽﾄｯﾊﾟｰ 抜 SOL
2426  LD      M663  ; 出口部 ｽﾄｯﾊﾟｰ 入
      ANI     Y2B6  ; 出口部 ｽﾄｯﾊﾟｰ 抜 SOL
      OUT     Y2B7  ; 出口部 ｽﾄｯﾊﾟｰ 入 SOL
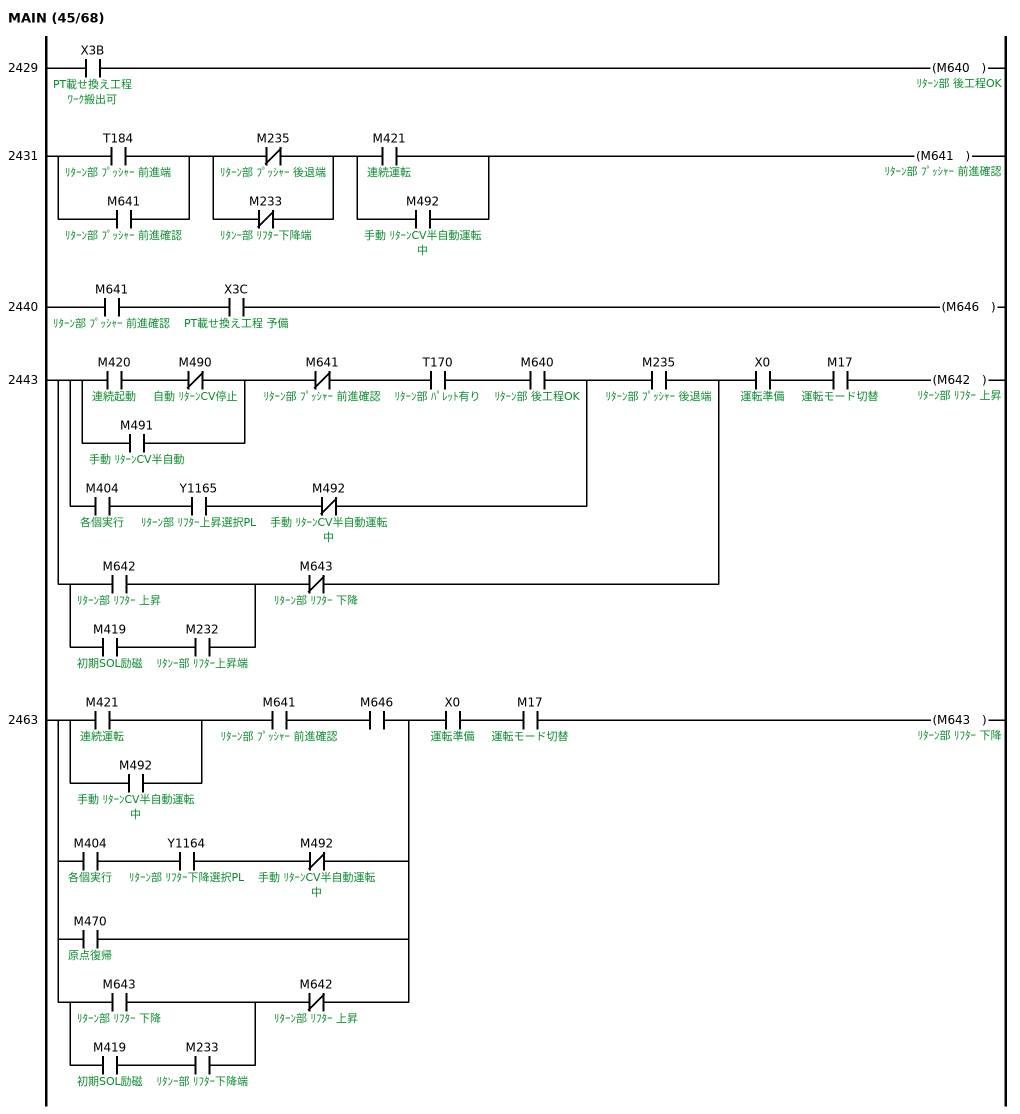
2429  LD      X3B  ; PT載せ換え工程 ﾜｰｸ搬出可
      OUT     M640  ; ﾘﾀｰﾝ部 後工程OK
2431  LD      T184  ; ﾘﾀｰﾝ部 ﾌﾟｯｼｬｰ 前進端
      OR      M641  ; ﾘﾀｰﾝ部 ﾌﾟｯｼｬｰ 前進確認
      LDI     M235  ; ﾘﾀｰﾝ部 ﾌﾟｯｼｬｰ 後退端
      ORI     M233  ; ﾘﾀﾝｰ部 ﾘﾌﾀｰ下降端
      ANB
      LD      M421  ; 連続運転
      OR      M492  ; 手動 ﾘﾀｰﾝCV半自動運転中
      ANB
      OUT     M641  ; ﾘﾀｰﾝ部 ﾌﾟｯｼｬｰ 前進確認
2440  LD      M641  ; ﾘﾀｰﾝ部 ﾌﾟｯｼｬｰ 前進確認
      AND     X3C  ; PT載せ換え工程 予備
      OUT     M646
2443  LD      M420  ; 連続起動
      ANI     M490  ; 自動 ﾘﾀｰﾝCV停止
      OR      M491  ; 手動 ﾘﾀｰﾝCV半自動
      ANI     M641  ; ﾘﾀｰﾝ部 ﾌﾟｯｼｬｰ 前進確認
      AND     T170  ; ﾘﾀｰﾝ部 ﾊﾟﾚｯﾄ有り
      AND     M640  ; ﾘﾀｰﾝ部 後工程OK
      LD      M404  ; 各個実行
      AND     Y1165  ; ﾘﾀｰﾝ部 ﾘﾌﾀｰ上昇選択PL
      ANI     M492  ; 手動 ﾘﾀｰﾝCV半自動運転中
      ORB
      AND     M235  ; ﾘﾀｰﾝ部 ﾌﾟｯｼｬｰ 後退端
      LD      M642  ; ﾘﾀｰﾝ部 ﾘﾌﾀｰ 上昇
      LD      M419  ; 初期SOL励磁
      AND     M232  ; ﾘﾀﾝｰ部 ﾘﾌﾀｰ上昇端
      ORB
      ANI     M643  ; ﾘﾀｰﾝ部 ﾘﾌﾀｰ 下降
      ORB
      AND     X0  ; 運転準備
      AND     M17  ; 運転モード切替
      OUT     M642  ; ﾘﾀｰﾝ部 ﾘﾌﾀｰ 上昇
2463  LD      M421  ; 連続運転
      OR      M492  ; 手動 ﾘﾀｰﾝCV半自動運転中
      AND     M641  ; ﾘﾀｰﾝ部 ﾌﾟｯｼｬｰ 前進確認
      AND     M646
      LD      M404  ; 各個実行
      AND     Y1164  ; ﾘﾀｰﾝ部 ﾘﾌﾀｰ下降選択PL
      ANI     M492  ; 手動 ﾘﾀｰﾝCV半自動運転中
      ORB
      OR      M470  ; 原点復帰
      LD      M643  ; ﾘﾀｰﾝ部 ﾘﾌﾀｰ 下降
      LD      M419  ; 初期SOL励磁
      AND     M233  ; ﾘﾀﾝｰ部 ﾘﾌﾀｰ下降端
      ORB
      ANI     M642  ; ﾘﾀｰﾝ部 ﾘﾌﾀｰ 上昇
      ORB
      AND     X0  ; 運転準備
      AND     M17  ; 運転モード切替
      OUT     M643  ; ﾘﾀｰﾝ部 ﾘﾌﾀｰ 下降
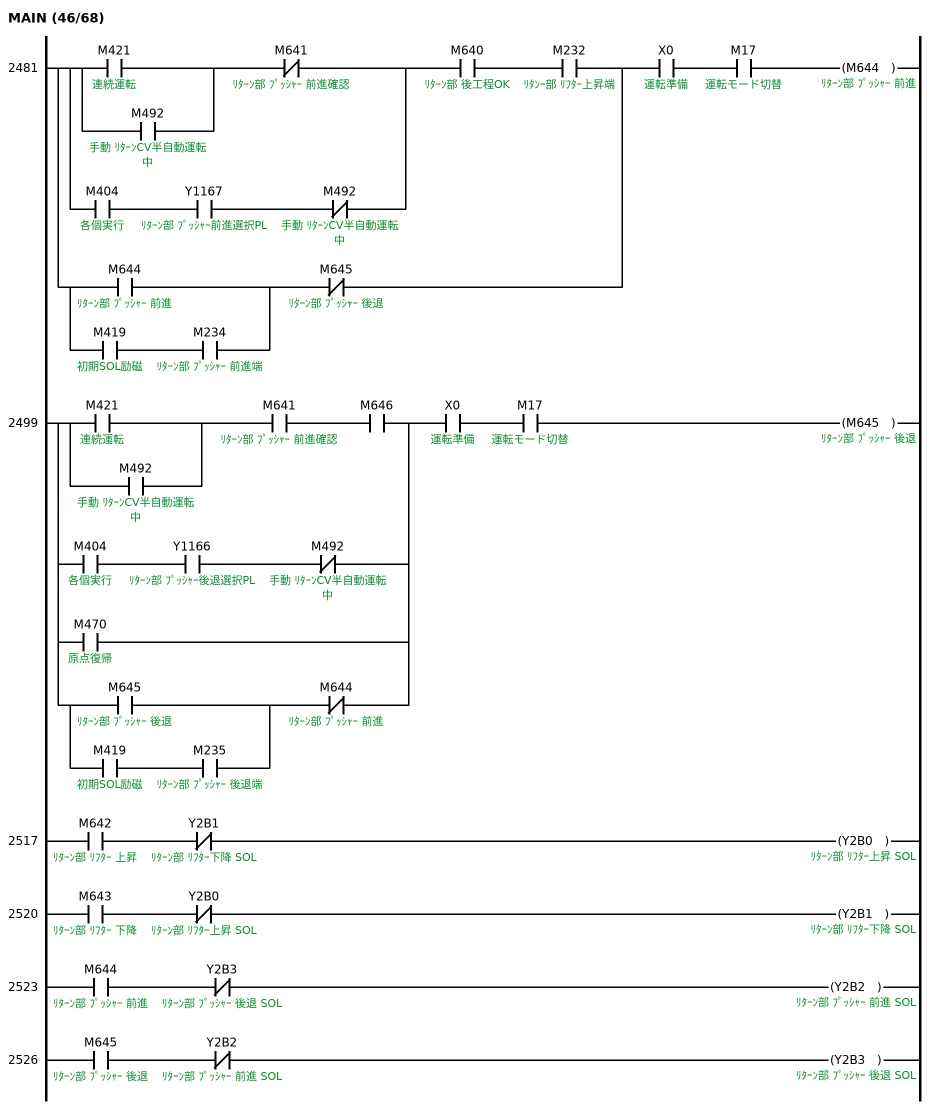
2481  LD      M421  ; 連続運転
      OR      M492  ; 手動 ﾘﾀｰﾝCV半自動運転中
      ANI     M641  ; ﾘﾀｰﾝ部 ﾌﾟｯｼｬｰ 前進確認
      LD      M404  ; 各個実行
      AND     Y1167  ; ﾘﾀｰﾝ部 ﾌﾟｯｼｬｰ前進選択PL
      ANI     M492  ; 手動 ﾘﾀｰﾝCV半自動運転中
      ORB
      AND     M640  ; ﾘﾀｰﾝ部 後工程OK
      AND     M232  ; ﾘﾀﾝｰ部 ﾘﾌﾀｰ上昇端
      LD      M644  ; ﾘﾀｰﾝ部 ﾌﾟｯｼｬｰ 前進
      LD      M419  ; 初期SOL励磁
      AND     M234  ; ﾘﾀｰﾝ部 ﾌﾟｯｼｬｰ 前進端
      ORB
      ANI     M645  ; ﾘﾀｰﾝ部 ﾌﾟｯｼｬｰ 後退
      ORB
      AND     X0  ; 運転準備
      AND     M17  ; 運転モード切替
      OUT     M644  ; ﾘﾀｰﾝ部 ﾌﾟｯｼｬｰ 前進
2499  LD      M421  ; 連続運転
      OR      M492  ; 手動 ﾘﾀｰﾝCV半自動運転中
      AND     M641  ; ﾘﾀｰﾝ部 ﾌﾟｯｼｬｰ 前進確認
      AND     M646
      LD      M404  ; 各個実行
      AND     Y1166  ; ﾘﾀｰﾝ部 ﾌﾟｯｼｬｰ後退選択PL
      ANI     M492  ; 手動 ﾘﾀｰﾝCV半自動運転中
      ORB
      OR      M470  ; 原点復帰
      LD      M645  ; ﾘﾀｰﾝ部 ﾌﾟｯｼｬｰ 後退
      LD      M419  ; 初期SOL励磁
      AND     M235  ; ﾘﾀｰﾝ部 ﾌﾟｯｼｬｰ 後退端
      ORB
      ANI     M644  ; ﾘﾀｰﾝ部 ﾌﾟｯｼｬｰ 前進
      ORB
      AND     X0  ; 運転準備
      AND     M17  ; 運転モード切替
      OUT     M645  ; ﾘﾀｰﾝ部 ﾌﾟｯｼｬｰ 後退
2517  LD      M642  ; ﾘﾀｰﾝ部 ﾘﾌﾀｰ 上昇
      ANI     Y2B1  ; ﾘﾀｰﾝ部 ﾘﾌﾀｰ下降 SOL
      OUT     Y2B0  ; ﾘﾀｰﾝ部 ﾘﾌﾀｰ上昇 SOL
2520  LD      M643  ; ﾘﾀｰﾝ部 ﾘﾌﾀｰ 下降
      ANI     Y2B0  ; ﾘﾀｰﾝ部 ﾘﾌﾀｰ上昇 SOL
      OUT     Y2B1  ; ﾘﾀｰﾝ部 ﾘﾌﾀｰ下降 SOL
2523  LD      M644  ; ﾘﾀｰﾝ部 ﾌﾟｯｼｬｰ 前進
      ANI     Y2B3  ; ﾘﾀｰﾝ部 ﾌﾟｯｼｬｰ 後退 SOL
      OUT     Y2B2  ; ﾘﾀｰﾝ部 ﾌﾟｯｼｬｰ 前進 SOL
2526  LD      M645  ; ﾘﾀｰﾝ部 ﾌﾟｯｼｬｰ 後退
      ANI     Y2B2  ; ﾘﾀｰﾝ部 ﾌﾟｯｼｬｰ 前進 SOL
      OUT     Y2B3  ; ﾘﾀｰﾝ部 ﾌﾟｯｼｬｰ 後退 SOL
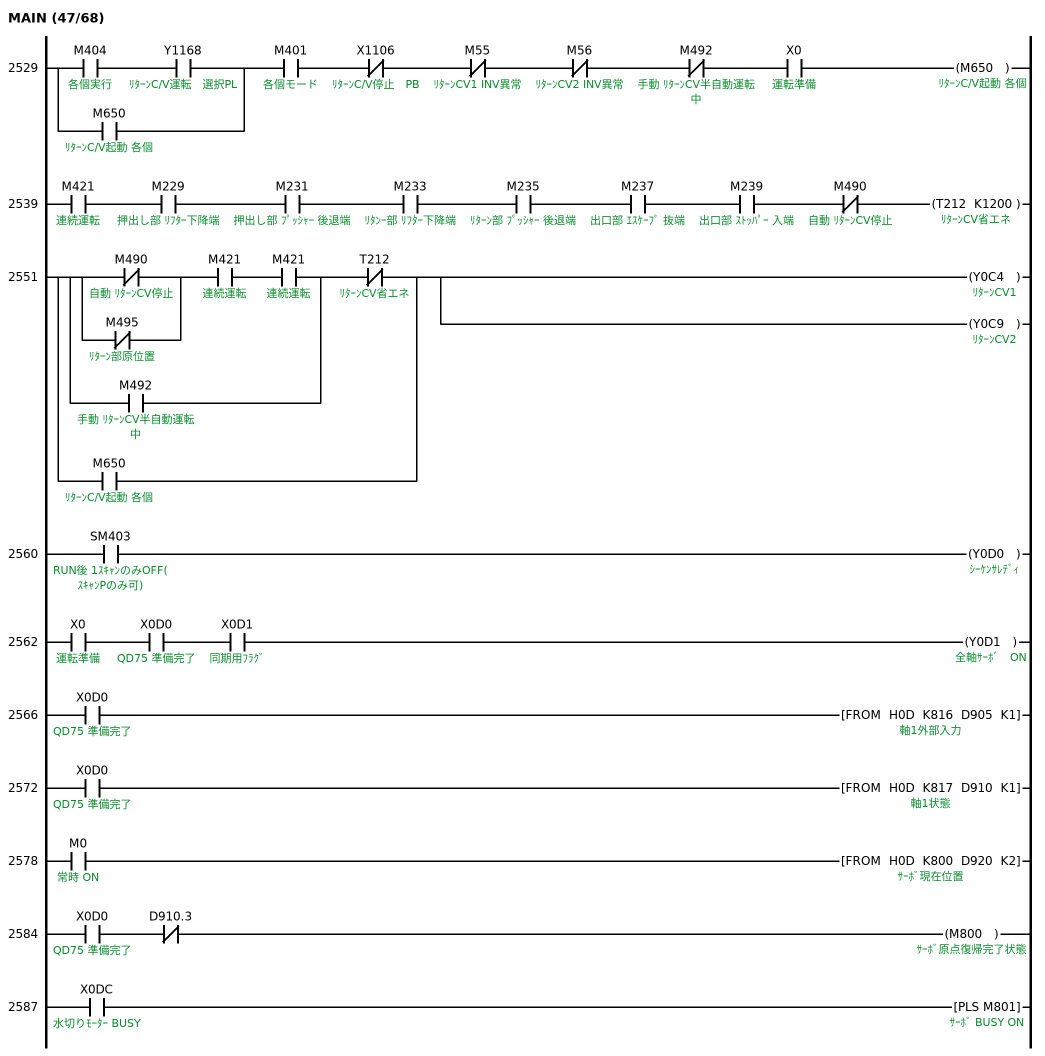
2529  LD      M404  ; 各個実行
      AND     Y1168  ; ﾘﾀｰﾝC/V運転　選択PL
      OR      M650  ; ﾘﾀｰﾝC/V起動 各個
      AND     M401  ; 各個モード
      ANI     X1106  ; ﾘﾀｰﾝC/V停止　PB
      ANI     M55  ; ﾘﾀｰﾝCV1 INV異常
      ANI     M56  ; ﾘﾀｰﾝCV2 INV異常
      ANI     M492  ; 手動 ﾘﾀｰﾝCV半自動運転中
      AND     X0  ; 運転準備
      OUT     M650  ; ﾘﾀｰﾝC/V起動 各個
2539  LD      M421  ; 連続運転
      AND     M229  ; 押出し部 ﾘﾌﾀｰ下降端
      AND     M231  ; 押出し部 ﾌﾟｯｼｬｰ 後退端
      AND     M233  ; ﾘﾀﾝｰ部 ﾘﾌﾀｰ下降端
      AND     M235  ; ﾘﾀｰﾝ部 ﾌﾟｯｼｬｰ 後退端
      AND     M237  ; 出口部 ｴｽｹｰﾌﾟ 抜端
      AND     M239  ; 出口部 ｽﾄｯﾊﾟｰ 入端
      ANI     M490  ; 自動 ﾘﾀｰﾝCV停止
      OUT     T212 K1200  ; ﾘﾀｰﾝCV省エネ
2551  LDI     M490  ; 自動 ﾘﾀｰﾝCV停止
      ORI     M495  ; ﾘﾀｰﾝ部原位置
      AND     M421  ; 連続運転
      AND     M421  ; 連続運転
      OR      M492  ; 手動 ﾘﾀｰﾝCV半自動運転中
      ANI     T212  ; ﾘﾀｰﾝCV省エネ
      OR      M650  ; ﾘﾀｰﾝC/V起動 各個
      OUT     Y0C4  ; ﾘﾀｰﾝCV1
      OUT     Y0C9  ; ﾘﾀｰﾝCV2
2560  LD      SM403  ; RUN後 1ｽｷｬﾝのみOFF(ｽｷｬﾝPのみ可)
      OUT     Y0D0  ; ｼｰｹﾝｻﾚﾃﾞｨ
2562  LD      X0  ; 運転準備
      AND     X0D0  ; QD75 準備完了
      AND     X0D1  ; 同期用ﾌﾗｸﾞ
      OUT     Y0D1  ; 全軸ｻｰﾎﾞ　ON
2566  LD      X0D0  ; QD75 準備完了
      FROM    H0D K816 D905 K1  ; 軸1外部入力
2572  LD      X0D0  ; QD75 準備完了
      FROM    H0D K817 D910 K1  ; 軸1状態
2578  LD      M0  ; 常時 ON
      FROM    H0D K800 D920 K2  ; ｻｰﾎﾞ現在位置
2584  LD      X0D0  ; QD75 準備完了
      ANI     D910.3
      OUT     M800  ; ｻｰﾎﾞ原点復帰完了状態
2587  LD      X0DC  ; 水切りﾓｰﾀｰ BUSY
      PLS     M801  ; ｻｰﾎﾞ BUSY ON
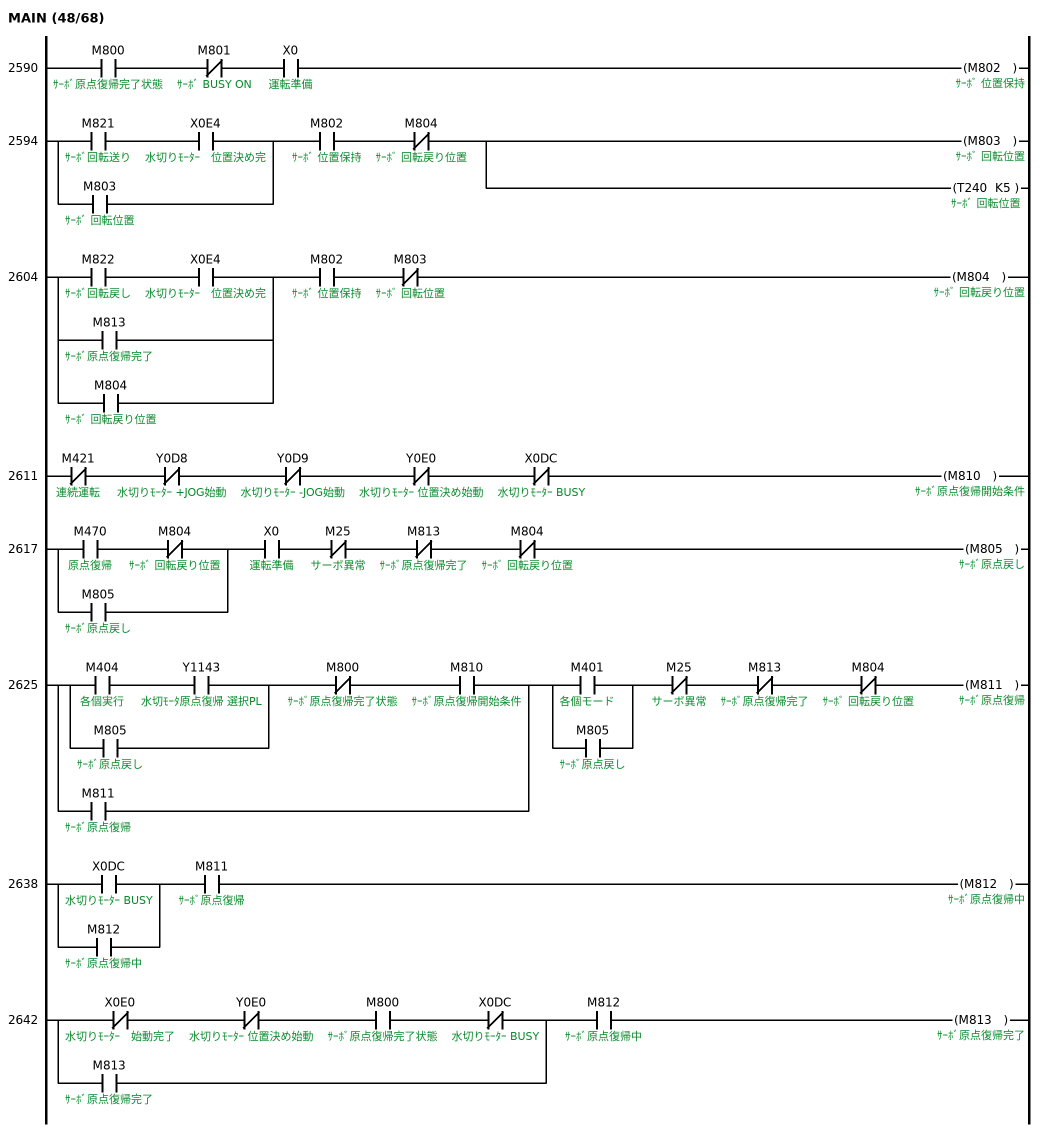
2590  LD      M800  ; ｻｰﾎﾞ原点復帰完了状態
      ANI     M801  ; ｻｰﾎﾞ BUSY ON
      AND     X0  ; 運転準備
      OUT     M802  ; ｻｰﾎﾞ 位置保持
2594  LD      M821  ; ｻｰﾎﾞ回転送り
      AND     X0E4  ; 水切りﾓｰﾀｰ　位置決め完
      OR      M803  ; ｻｰﾎﾞ 回転位置
      AND     M802  ; ｻｰﾎﾞ 位置保持
      ANI     M804  ; ｻｰﾎﾞ 回転戻り位置
      OUT     M803  ; ｻｰﾎﾞ 回転位置
      OUT     T240 K5  ; ｻｰﾎﾞ 回転位置
2604  LD      M822  ; ｻｰﾎﾞ回転戻し
      AND     X0E4  ; 水切りﾓｰﾀｰ　位置決め完
      OR      M813  ; ｻｰﾎﾞ原点復帰完了
      OR      M804  ; ｻｰﾎﾞ 回転戻り位置
      AND     M802  ; ｻｰﾎﾞ 位置保持
      ANI     M803  ; ｻｰﾎﾞ 回転位置
      OUT     M804  ; ｻｰﾎﾞ 回転戻り位置
2611  LDI     M421  ; 連続運転
      ANI     Y0D8  ; 水切りﾓｰﾀｰ +JOG始動
      ANI     Y0D9  ; 水切りﾓｰﾀｰ -JOG始動
      ANI     Y0E0  ; 水切りﾓｰﾀｰ 位置決め始動
      ANI     X0DC  ; 水切りﾓｰﾀｰ BUSY
      OUT     M810  ; ｻｰﾎﾞ原点復帰開始条件
2617  LD      M470  ; 原点復帰
      ANI     M804  ; ｻｰﾎﾞ 回転戻り位置
      OR      M805  ; ｻｰﾎﾞ原点戻し
      AND     X0  ; 運転準備
      ANI     M25  ; サーボ異常
      ANI     M813  ; ｻｰﾎﾞ原点復帰完了
      ANI     M804  ; ｻｰﾎﾞ 回転戻り位置
      OUT     M805  ; ｻｰﾎﾞ原点戻し
2625  LD      M404  ; 各個実行
      AND     Y1143  ; 水切ﾓｰﾀ原点復帰 選択PL
      OR      M805  ; ｻｰﾎﾞ原点戻し
      ANI     M800  ; ｻｰﾎﾞ原点復帰完了状態
      AND     M810  ; ｻｰﾎﾞ原点復帰開始条件
      OR      M811  ; ｻｰﾎﾞ原点復帰
      LD      M401  ; 各個モード
      OR      M805  ; ｻｰﾎﾞ原点戻し
      ANB
      ANI     M25  ; サーボ異常
      ANI     M813  ; ｻｰﾎﾞ原点復帰完了
      ANI     M804  ; ｻｰﾎﾞ 回転戻り位置
      OUT     M811  ; ｻｰﾎﾞ原点復帰
2638  LD      X0DC  ; 水切りﾓｰﾀｰ BUSY
      OR      M812  ; ｻｰﾎﾞ原点復帰中
      AND     M811  ; ｻｰﾎﾞ原点復帰
      OUT     M812  ; ｻｰﾎﾞ原点復帰中
2642  LDI     X0E0  ; 水切りﾓｰﾀｰ　始動完了
      ANI     Y0E0  ; 水切りﾓｰﾀｰ 位置決め始動
      AND     M800  ; ｻｰﾎﾞ原点復帰完了状態
      ANI     X0DC  ; 水切りﾓｰﾀｰ BUSY
      OR      M813  ; ｻｰﾎﾞ原点復帰完了
      AND     M812  ; ｻｰﾎﾞ原点復帰中
      OUT     M813  ; ｻｰﾎﾞ原点復帰完了
